LIN {X 0,Y 417.094,Z 395.374,A -85,B 0,C 180,E1 -10165.652,E2 -10165.652} C_VEL
LIN {X 0,Y 417.167,Z 397.871,A -85,B 0,C 180,E1 -10167.103,E2 -10167.103} C_VEL
LIN {X 0,Y 417.136,Z 398.972,A -85,B 0,C 180,E1 -10168.069,E2 -10168.069} C_VEL
LIN {X 0,Y 417.115,Z 399.643,A -85,B 0,C 180,E1 -10169.035,E2 -10169.035} C_VEL
LIN {X 0,Y 417.13,Z 399.91,A -85,B 0,C 180,E1 -10170,E2 -10170} C_VEL
LIN {X 0,Y 417.089,Z 399.765,A -85,B 0,C 180,E1 -10170.966,E2 -10170.966} C_VEL
LIN {X 0,Y 417.118,Z 399.169,A -85,B 0,C 180,E1 -10171.931,E2 -10171.931} C_VEL
LIN {X 0,Y 417.132,Z 398.154,A -85,B 0,C 180,E1 -10172.898,E2 -10172.898} C_VEL
LIN {X 0,Y 417.056,Z 396.723,A -85,B 0,C 180,E1 -10173.865,E2 -10173.865} C_VEL
LIN {X 0,Y 417.128,Z 393.73,A -85,B 0,C 180,E1 -10175.317,E2 -10175.317} C_VEL
LIN {X 0,Y 417.159,Z 389.667,A -85,B 0,C 180,E1 -10176.773,E2 -10176.773} C_VEL
LIN {X 0,Y 417.432,Z 383.444,A -85,B 0,C 180,E1 -10178.472,E2 -10178.472} C_VEL
LIN {X 0,Y 417.77,Z 376.616,A -85,B 0,C 180,E1 -10179.93,E2 -10179.93} C_VEL
LIN {X 0,Y 418.327,Z 368.161,A -85,B 0,C 180,E1 -10181.385,E2 -10181.385} C_VEL
LIN {X 0,Y 418.871,Z 359.55,A -85,B 0,C 180,E1 -10182.599,E2 -10182.599} C_VEL
LIN {X 0,Y 419.553,Z 349.191,A -85,B 0,C 180,E1 -10183.785,E2 -10183.785} C_VEL
LIN {X 0,Y 420.452,Z 337.073,A -85,B 0,C 180,E1 -10184.892,E2 -10184.892} C_VEL
LIN {X 0,Y 421.245,Z 325.274,A -85,B 0,C 180,E1 -10185.731,E2 -10185.731} C_VEL
LIN {X 0,Y 422,Z 311.923,A -85,B 0,C 180,E1 -10186.447,E2 -10186.447} C_VEL
LIN {X 0,Y 422.679,Z 299.417,A -85,B 0,C 180,E1 -10186.917,E2 -10186.917} C_VEL
LIN {X 0,Y 423.066,Z 283.977,A -85,B 0,C 180,E1 -10187.274,E2 -10187.274} C_VEL
LIN {X 0,Y 424.143,Z 213.784,A -85,B 0,C 180,E1 -10188.664,E2 -10188.664} C_VEL
LIN {X 0,Y 421.797,Z 196.296,A -85,B 0,C 180,E1 -10189.167,E2 -10189.167} C_VEL
LIN {X 0,Y 419.76,Z 184.639,A -85,B 0,C 180,E1 -10189.564,E2 -10189.564} C_VEL
LIN {X 0,Y 421.003,Z 163.827,A -85,B 0,C 180,E1 -10193.343,E2 -10193.343} C_VEL
LIN {X 0,Y 421.708,Z 152.632,A -85,B 0,C 180,E1 -10195.413,E2 -10195.413} C_VEL
LIN {X 0,Y 419.796,Z 142.649,A -85,B 0,C 180,E1 -10197.464,E2 -10197.464} C_VEL
LIN {X 0,Y 418.315,Z 136.387,A -85,B 0,C 180,E1 -10198.855,E2 -10198.855} C_VEL
LIN {X 0,Y 418.249,Z 136.39,A -85,B 0,C 180,E1 -10202.528,E2 -10202.528} C_VEL
LIN {X 0,Y 418.263,Z 136.385,A -85,B 0,C 180,E1 -10204.841,E2 -10204.841} C_VEL
LIN {X 0,Y 418.261,Z 136.386,A -85,B 0,C 180,E1 -10208.441,E2 -10208.441} C_VEL
LIN {X 0,Y 418.227,Z 136.388,A -85,B 0,C 180,E1 -10210.948,E2 -10210.948} C_VEL
LIN {X 0,Y 418.214,Z 136.391,A -85,B 0,C 180,E1 -10213.729,E2 -10213.729} C_VEL
LIN {X 0,Y 418.213,Z 136.388,A -85,B 0,C 180,E1 -10216.449,E2 -10216.449} C_VEL
LIN {X 0,Y 418.226,Z 136.384,A -85,B 0,C 180,E1 -10219.13,E2 -10219.13} C_VEL
LIN {X 0,Y 418.229,Z 136.385,A -85,B 0,C 180,E1 -10222.167,E2 -10222.167} C_VEL
LIN {X 0,Y 418.267,Z 136.382,A -85,B 0,C 180,E1 -10225.42,E2 -10225.42} C_VEL
LIN {X 0,Y 418.214,Z 136.384,A -85,B 0,C 180,E1 -10228.604,E2 -10228.604} C_VEL
LIN {X 0,Y 418.295,Z 136.38,A -85,B 0,C 180,E1 -10231.937,E2 -10231.937} C_VEL
LIN {X 0,Y 418.293,Z 136.38,A -85,B 0,C 180,E1 -10235.163,E2 -10235.163} C_VEL
LIN {X 0,Y 418.237,Z 136.385,A -85,B 0,C 180,E1 -10238.303,E2 -10238.303} C_VEL
LIN {X 0,Y 418.278,Z 136.38,A -85,B 0,C 180,E1 -10241.383,E2 -10241.383} C_VEL
LIN {X 0,Y 418.304,Z 136.377,A -85,B 0,C 180,E1 -10244.406,E2 -10244.406} C_VEL
LIN {X 0,Y 418.359,Z 136.373,A -85,B 0,C 180,E1 -10247.385,E2 -10247.385} C_VEL
LIN {X 0,Y 418.341,Z 136.376,A -85,B 0,C 180,E1 -10250.328,E2 -10250.328} C_VEL
LIN {X 0,Y 418.463,Z 136.363,A -85,B 0,C 180,E1 -10253.248,E2 -10253.248} C_VEL
LIN {X 0,Y 418.336,Z 136.378,A -85,B 0,C 180,E1 -10255.181,E2 -10255.181} C_VEL
LIN {X 0,Y 418.543,Z 136.354,A -85,B 0,C 180,E1 -10258.075,E2 -10258.075} C_VEL
LIN {X 0,Y 418.669,Z 136.335,A -85,B 0,C 180,E1 -10260,E2 -10260} C_VEL
LIN {X 0,Y 418.49,Z 136.36,A -85,B 0,C 180,E1 -10262.887,E2 -10262.887} C_VEL
LIN {X 0,Y 418.393,Z 136.563,A -85,B 0,C 180,E1 -10263.43,E2 -10263.43} C_VEL
LIN {X 0,Y 420.352,Z 145.319,A -85,B 0,C 180,E1 -10265.546,E2 -10265.546} C_VEL
LIN {X 0,Y 422.812,Z 152.93,A -85,B 0,C 180,E1 -10265.873,E2 -10265.873} C_VEL
LIN {X 0,Y 425.067,Z 163.368,A -85,B 0,C 180,E1 -10266.228,E2 -10266.228} C_VEL
LIN {X 0,Y 423.251,Z 252.714,A -85,B 0,C 180,E1 -10268.023,E2 -10268.023} C_VEL
LIN {X 0,Y 422.865,Z 266.764,A -85,B 0,C 180,E1 -10268.512,E2 -10268.512} C_VEL
LIN {X 0,Y 422.412,Z 278.341,A -85,B 0,C 180,E1 -10269.094,E2 -10269.094} C_VEL
LIN {X 0,Y 421.766,Z 290.403,A -85,B 0,C 180,E1 -10269.903,E2 -10269.903} C_VEL
LIN {X 0,Y 421.007,Z 302.463,A -85,B 0,C 180,E1 -10270.946,E2 -10270.946} C_VEL
LIN {X 0,Y 420.288,Z 312.69,A -85,B 0,C 180,E1 -10272.065,E2 -10272.065} C_VEL
LIN {X 0,Y 419.627,Z 321.922,A -85,B 0,C 180,E1 -10273.314,E2 -10273.314} C_VEL
LIN {X 0,Y 419.021,Z 329.545,A -85,B 0,C 180,E1 -10274.571,E2 -10274.571} C_VEL
LIN {X 0,Y 418.437,Z 336.998,A -85,B 0,C 180,E1 -10276.089,E2 -10276.089} C_VEL
LIN {X 0,Y 418.001,Z 342.862,A -85,B 0,C 180,E1 -10277.616,E2 -10277.616} C_VEL
LIN {X 0,Y 417.659,Z 347.251,A -85,B 0,C 180,E1 -10279.083,E2 -10279.083} C_VEL
LIN {X 0,Y 417.369,Z 350.82,A -85,B 0,C 180,E1 -10280.708,E2 -10280.708} C_VEL
LIN {X 0,Y 417.184,Z 352.874,A -85,B 0,C 180,E1 -10282.097,E2 -10282.097} C_VEL
LIN {X 0,Y 417.034,Z 354.234,A -85,B 0,C 180,E1 -10283.857,E2 -10283.857} C_VEL
LIN {X 0,Y 417.033,Z 354.402,A -85,B 0,C 180,E1 -10284.917,E2 -10284.917} C_VEL
LIN {X 0,Y 417.067,Z 353.497,A -85,B 0,C 180,E1 -10286.733,E2 -10286.733} C_VEL
LIN {X 0,Y 417.126,Z 351.798,A -85,B 0,C 180,E1 -10288.148,E2 -10288.148} C_VEL
LIN {X 0,Y 417.344,Z 348.667,A -85,B 0,C 180,E1 -10289.786,E2 -10289.786} C_VEL
LIN {X 0,Y 417.543,Z 344.141,A -85,B 0,C 180,E1 -10291.452,E2 -10291.452} C_VEL
LIN {X 0,Y 417.849,Z 339.491,A -85,B 0,C 180,E1 -10292.757,E2 -10292.757} C_VEL
LIN {X 0,Y 418.25,Z 332.297,A -85,B 0,C 180,E1 -10294.364,E2 -10294.364} C_VEL
LIN {X 0,Y 418.73,Z 324.93,A -85,B 0,C 180,E1 -10295.679,E2 -10295.679} C_VEL
LIN {X 0,Y 419.225,Z 316.571,A -85,B 0,C 180,E1 -10296.906,E2 -10296.906} C_VEL
LIN {X 0,Y 419.837,Z 306.507,A -85,B 0,C 180,E1 -10298.115,E2 -10298.115} C_VEL
LIN {X 0,Y 420.414,Z 296,A -85,B 0,C 180,E1 -10299.128,E2 -10299.128} C_VEL
LIN {X 0,Y 420.983,Z 284.099,A -85,B 0,C 180,E1 -10300.04,E2 -10300.04} C_VEL
LIN {X 0,Y 421.48,Z 272.646,A -85,B 0,C 180,E1 -10300.719,E2 -10300.719} C_VEL
LIN {X 0,Y 421.837,Z 259.788,A -85,B 0,C 180,E1 -10301.279,E2 -10301.279} C_VEL
LIN {X 0,Y 422.128,Z 246.612,A -85,B 0,C 180,E1 -10301.649,E2 -10301.649} C_VEL
LIN {X 0,Y 423.408,Z 161.415,A -85,B 0,C 180,E1 -10303.267,E2 -10303.267} C_VEL
LIN {X 0,Y 419.546,Z 143.216,A -85,B 0,C 180,E1 -10303.8,E2 -10303.8} C_VEL
LIN {X 0,Y 418.289,Z 136.384,A -85,B 0,C 180,E1 -10305.466,E2 -10305.466} C_VEL
LIN {X 0,Y 418.222,Z 136.387,A -85,B 0,C 180,E1 -10309.13,E2 -10309.13} C_VEL
LIN {X 0,Y 418.225,Z 136.387,A -85,B 0,C 180,E1 -10312.167,E2 -10312.167} C_VEL
LIN {X 0,Y 418.263,Z 136.386,A -85,B 0,C 180,E1 -10315.42,E2 -10315.42} C_VEL
LIN {X 0,Y 418.21,Z 136.387,A -85,B 0,C 180,E1 -10318.603,E2 -10318.603} C_VEL
LIN {X 0,Y 418.291,Z 136.379,A -85,B 0,C 180,E1 -10321.936,E2 -10321.936} C_VEL
LIN {X 0,Y 418.289,Z 136.382,A -85,B 0,C 180,E1 -10325.162,E2 -10325.162} C_VEL
LIN {X 0,Y 418.276,Z 136.378,A -85,B 0,C 180,E1 -10326.002,E2 -10326.002} C_VEL
LIN {X 0,Y 417.636,Z 136.462,A -85,B 0,C 180,E1 -10326.805,E2 -10326.805} C_VEL
LIN {X 0,Y 414.786,Z 136.814,A -85,B 0,C 180,E1 -10328.11,E2 -10328.11} C_VEL
LIN {X 0,Y 412.35,Z 137.123,A -85,B 0,C 180,E1 -10329.164,E2 -10329.164} C_VEL
LIN {X 0,Y 411.294,Z 137.249,A -85,B 0,C 180,E1 -10329.978,E2 -10329.978} C_VEL
LIN {X 0,Y 411.204,Z 137.26,A -85,B 0,C 180,E1 -10330.254,E2 -10330.254} C_VEL
LIN {X 0,Y 411.262,Z 137.259,A -85,B 0,C 180,E1 -10333.131,E2 -10333.131} C_VEL
LIN {X 0,Y 411.304,Z 137.252,A -85,B 0,C 180,E1 -10336.895,E2 -10336.895} C_VEL
LIN {X 0,Y 411.292,Z 137.249,A -85,B 0,C 180,E1 -10340.161,E2 -10340.161} C_VEL
LIN {X 0,Y 411.45,Z 137.234,A -85,B 0,C 180,E1 -10343.133,E2 -10343.133} C_VEL
LIN {X 0,Y 411.308,Z 137.252,A -85,B 0,C 180,E1 -10345.099,E2 -10345.099} C_VEL
LIN {X 0,Y 411.513,Z 137.221,A -85,B 0,C 180,E1 -10348.042,E2 -10348.042} C_VEL
LIN {X 0,Y 411.641,Z 137.205,A -85,B 0,C 180,E1 -10350,E2 -10350} C_VEL
LIN {X 0,Y 411.463,Z 137.232,A -85,B 0,C 180,E1 -10352.937,E2 -10352.937} C_VEL
LIN {X 0,Y 411.45,Z 137.234,A -85,B 0,C 180,E1 -10356.867,E2 -10356.867} C_VEL
LIN {X 0,Y 411.291,Z 137.249,A -85,B 0,C 180,E1 -10359.838,E2 -10359.838} C_VEL
LIN {X 0,Y 411.303,Z 137.249,A -85,B 0,C 180,E1 -10363.104,E2 -10363.104} C_VEL
LIN {X 0,Y 411.26,Z 137.255,A -85,B 0,C 180,E1 -10366.869,E2 -10366.869} C_VEL
LIN {X 0,Y 411.228,Z 137.259,A -85,B 0,C 180,E1 -10369.986,E2 -10369.986} C_VEL
LIN {X 0,Y 411.193,Z 137.261,A -85,B 0,C 180,E1 -10373.148,E2 -10373.148} C_VEL
LIN {X 0,Y 411.233,Z 137.262,A -85,B 0,C 180,E1 -10376.381,E2 -10376.381} C_VEL
LIN {X 0,Y 411.208,Z 137.261,A -85,B 0,C 180,E1 -10379.712,E2 -10379.712} C_VEL
LIN {X 0,Y 411.204,Z 137.26,A -85,B 0,C 180,E1 -10383.156,E2 -10383.156} C_VEL
LIN {X 0,Y 411.192,Z 137.263,A -85,B 0,C 180,E1 -10386.553,E2 -10386.553} C_VEL
LIN {X 0,Y 411.213,Z 137.263,A -85,B 0,C 180,E1 -10389.728,E2 -10389.728} C_VEL
LIN {X 0,Y 411.227,Z 137.257,A -85,B 0,C 180,E1 -10393.126,E2 -10393.126} C_VEL
LIN {X 0,Y 411.168,Z 137.271,A -85,B 0,C 180,E1 -10395.88,E2 -10395.88} C_VEL
LIN {X 0,Y 411.208,Z 137.263,A -85,B 0,C 180,E1 -10399.499,E2 -10399.499} C_VEL
LIN {X 0,Y 411.2,Z 137.263,A -85,B 0,C 180,E1 -10402.027,E2 -10402.027} C_VEL
LIN {X 0,Y 411.203,Z 137.266,A -85,B 0,C 180,E1 -10405.667,E2 -10405.667} C_VEL
LIN {X 0,Y 411.186,Z 137.265,A -85,B 0,C 180,E1 -10409.153,E2 -10409.153} C_VEL
LIN {X 0,Y 411.255,Z 137.253,A -85,B 0,C 180,E1 -10412.523,E2 -10412.523} C_VEL
LIN {X 0,Y 411.224,Z 137.26,A -85,B 0,C 180,E1 -10415.785,E2 -10415.785} C_VEL
LIN {X 0,Y 411.193,Z 137.264,A -85,B 0,C 180,E1 -10418.966,E2 -10418.966} C_VEL
LIN {X 0,Y 411.25,Z 137.254,A -85,B 0,C 180,E1 -10422.085,E2 -10422.085} C_VEL
LIN {X 0,Y 411.257,Z 137.26,A -85,B 0,C 180,E1 -10425.148,E2 -10425.148} C_VEL
LIN {X 0,Y 411.282,Z 137.25,A -85,B 0,C 180,E1 -10428.168,E2 -10428.168} C_VEL
LIN {X 0,Y 411.438,Z 137.231,A -85,B 0,C 180,E1 -10432.189,E2 -10432.189} C_VEL
LIN {X 0,Y 411.469,Z 137.227,A -85,B 0,C 180,E1 -10434.118,E2 -10434.118} C_VEL
LIN {X 0,Y 411.512,Z 137.221,A -85,B 0,C 180,E1 -10438.043,E2 -10438.043} C_VEL
LIN {X 0,Y 411.64,Z 137.205,A -85,B 0,C 180,E1 -10440,E2 -10440} C_VEL
LIN {X 0,Y 411.463,Z 137.233,A -85,B 0,C 180,E1 -10442.938,E2 -10442.938} C_VEL
LIN {X 0,Y 411.459,Z 137.233,A -85,B 0,C 180,E1 -10446.867,E2 -10446.867} C_VEL
LIN {X 0,Y 411.292,Z 137.249,A -85,B 0,C 180,E1 -10449.839,E2 -10449.839} C_VEL
LIN {X 0,Y 411.304,Z 137.249,A -85,B 0,C 180,E1 -10453.105,E2 -10453.105} C_VEL
LIN {X 0,Y 411.262,Z 137.255,A -85,B 0,C 180,E1 -10456.869,E2 -10456.869} C_VEL
LIN {X 0,Y 411.229,Z 137.259,A -85,B 0,C 180,E1 -10459.987,E2 -10459.987} C_VEL
LIN {X 0,Y 411.194,Z 137.261,A -85,B 0,C 180,E1 -10463.148,E2 -10463.148} C_VEL
LIN {X 0,Y 411.235,Z 137.262,A -85,B 0,C 180,E1 -10466.381,E2 -10466.381} C_VEL
LIN {X 0,Y 411.199,Z 137.262,A -85,B 0,C 180,E1 -10469.713,E2 -10469.713} C_VEL
LIN {X 0,Y 411.206,Z 137.259,A -85,B 0,C 180,E1 -10473.156,E2 -10473.156} C_VEL
LIN {X 0,Y 411.195,Z 137.263,A -85,B 0,C 180,E1 -10476.554,E2 -10476.554} C_VEL
LIN {X 0,Y 411.226,Z 137.261,A -85,B 0,C 180,E1 -10479.731,E2 -10479.731} C_VEL
LIN {X 0,Y 411.178,Z 137.263,A -85,B 0,C 180,E1 -10483.133,E2 -10483.133} C_VEL
LIN {X 0,Y 411.168,Z 137.271,A -85,B 0,C 180,E1 -10485.882,E2 -10485.882} C_VEL
LIN {X 0,Y 411.163,Z 137.265,A -85,B 0,C 180,E1 -10488.772,E2 -10488.772} C_VEL
LIN {X 0,Y 411.205,Z 137.266,A -85,B 0,C 180,E1 -10491.832,E2 -10491.832} C_VEL
LIN {X 0,Y 411.211,Z 137.26,A -85,B 0,C 180,E1 -10495.122,E2 -10495.122} C_VEL
LIN {X 0,Y 411.166,Z 137.269,A -85,B 0,C 180,E1 -10498.003,E2 -10498.003} C_VEL
LIN {X 0,Y 411.299,Z 137.404,A -85,B 0,C 180,E1 -10501.326,E2 -10501.326} C_VEL
LIN {X 0,Y 414.04,Z 150.868,A -85,B 0,C 180,E1 -10504.111,E2 -10504.111} C_VEL
LIN {X 0,Y 414.425,Z 154.951,A -85,B 0,C 180,E1 -10504.916,E2 -10504.916} C_VEL
LIN {X 0,Y 413.221,Z 172.954,A -85,B 0,C 180,E1 -10508.29,E2 -10508.29} C_VEL
LIN {X 0,Y 412.419,Z 187.182,A -85,B 0,C 180,E1 -10510.923,E2 -10510.923} C_VEL
LIN {X 0,Y 416.159,Z 215.844,A -85,B 0,C 180,E1 -10511.653,E2 -10511.653} C_VEL
LIN {X 0,Y 414.934,Z 296.264,A -85,B 0,C 180,E1 -10513.234,E2 -10513.234} C_VEL
LIN {X 0,Y 414.347,Z 310.436,A -85,B 0,C 180,E1 -10513.717,E2 -10513.717} C_VEL
LIN {X 0,Y 413.746,Z 323.086,A -85,B 0,C 180,E1 -10514.357,E2 -10514.357} C_VEL
LIN {X 0,Y 412.93,Z 335.573,A -85,B 0,C 180,E1 -10515.209,E2 -10515.209} C_VEL
LIN {X 0,Y 412.315,Z 346.811,A -85,B 0,C 180,E1 -10516.195,E2 -10516.195} C_VEL
LIN {X 0,Y 411.774,Z 355.924,A -85,B 0,C 180,E1 -10517.181,E2 -10517.181} C_VEL
LIN {X 0,Y 411.231,Z 365.272,A -85,B 0,C 180,E1 -10518.416,E2 -10518.416} C_VEL
LIN {X 0,Y 410.638,Z 374.356,A -85,B 0,C 180,E1 -10519.897,E2 -10519.897} C_VEL
LIN {X 0,Y 410.346,Z 381.654,A -85,B 0,C 180,E1 -10521.381,E2 -10521.381} C_VEL
LIN {X 0,Y 410.166,Z 386.569,A -85,B 0,C 180,E1 -10522.617,E2 -10522.617} C_VEL
LIN {X 0,Y 410.009,Z 391.307,A -85,B 0,C 180,E1 -10524.097,E2 -10524.097} C_VEL
LIN {X 0,Y 410.021,Z 394.891,A -85,B 0,C 180,E1 -10525.577,E2 -10525.577} C_VEL
LIN {X 0,Y 410.08,Z 397.415,A -85,B 0,C 180,E1 -10527.053,E2 -10527.053} C_VEL
LIN {X 0,Y 410.063,Z 398.546,A -85,B 0,C 180,E1 -10528.036,E2 -10528.036} C_VEL
LIN {X 0,Y 410.034,Z 399.229,A -85,B 0,C 180,E1 -10529.018,E2 -10529.018} C_VEL
LIN {X 0,Y 410.046,Z 399.509,A -85,B 0,C 180,E1 -10530,E2 -10530} C_VEL
LIN {X 0,Y 410.01,Z 399.378,A -85,B 0,C 180,E1 -10530.983,E2 -10530.983} C_VEL
LIN {X 0,Y 410.045,Z 398.803,A -85,B 0,C 180,E1 -10531.965,E2 -10531.965} C_VEL
LIN {X 0,Y 410.029,Z 397.798,A -85,B 0,C 180,E1 -10532.948,E2 -10532.948} C_VEL
LIN {X 0,Y 409.972,Z 396.378,A -85,B 0,C 180,E1 -10533.932,E2 -10533.932} C_VEL
LIN {X 0,Y 410.018,Z 393.403,A -85,B 0,C 180,E1 -10535.41,E2 -10535.41} C_VEL
LIN {X 0,Y 410.077,Z 389.358,A -85,B 0,C 180,E1 -10536.891,E2 -10536.891} C_VEL
LIN {X 0,Y 410.355,Z 383.175,A -85,B 0,C 180,E1 -10538.619,E2 -10538.619} C_VEL
LIN {X 0,Y 410.741,Z 376.38,A -85,B 0,C 180,E1 -10540.101,E2 -10540.101} C_VEL
LIN {X 0,Y 411.335,Z 367.962,A -85,B 0,C 180,E1 -10541.582,E2 -10541.582} C_VEL
LIN {X 0,Y 411.903,Z 359.384,A -85,B 0,C 180,E1 -10542.816,E2 -10542.816} C_VEL
LIN {X 0,Y 412.662,Z 348.874,A -85,B 0,C 180,E1 -10544.046,E2 -10544.046} C_VEL
LIN {X 0,Y 413.588,Z 337.088,A -85,B 0,C 180,E1 -10545.145,E2 -10545.145} C_VEL
LIN {X 0,Y 414.44,Z 325.483,A -85,B 0,C 180,E1 -10545.996,E2 -10545.996} C_VEL
LIN {X 0,Y 415.225,Z 312.334,A -85,B 0,C 180,E1 -10546.723,E2 -10546.723} C_VEL
LIN {X 0,Y 415.967,Z 299.323,A -85,B 0,C 180,E1 -10547.23,E2 -10547.23} C_VEL
LIN {X 0,Y 416.379,Z 284.262,A -85,B 0,C 180,E1 -10547.592,E2 -10547.592} C_VEL
LIN {X 0,Y 417.533,Z 214.569,A -85,B 0,C 180,E1 -10549.008,E2 -10549.008} C_VEL
LIN {X 0,Y 415.28,Z 197.666,A -85,B 0,C 180,E1 -10549.512,E2 -10549.512} C_VEL
LIN {X 0,Y 412.933,Z 184.186,A -85,B 0,C 180,E1 -10549.976,E2 -10549.976} C_VEL
LIN {X 0,Y 414.158,Z 164.617,A -85,B 0,C 180,E1 -10553.602,E2 -10553.602} C_VEL
LIN {X 0,Y 414.86,Z 154.266,A -85,B 0,C 180,E1 -10555.546,E2 -10555.546} C_VEL
LIN {X 0,Y 412.871,Z 143.922,A -85,B 0,C 180,E1 -10557.728,E2 -10557.728} C_VEL
LIN {X 0,Y 411.237,Z 137.268,A -85,B 0,C 180,E1 -10559.211,E2 -10559.211} C_VEL
LIN {X 0,Y 411.169,Z 137.273,A -85,B 0,C 180,E1 -10561.997,E2 -10561.997} C_VEL
LIN {X 0,Y 411.214,Z 137.263,A -85,B 0,C 180,E1 -10564.879,E2 -10564.879} C_VEL
LIN {X 0,Y 411.211,Z 137.265,A -85,B 0,C 180,E1 -10568.169,E2 -10568.169} C_VEL
LIN {X 0,Y 411.168,Z 137.268,A -85,B 0,C 180,E1 -10571.228,E2 -10571.228} C_VEL
LIN {X 0,Y 411.179,Z 137.266,A -85,B 0,C 180,E1 -10574.49,E2 -10574.49} C_VEL
LIN {X 0,Y 411.181,Z 137.262,A -85,B 0,C 180,E1 -10578.195,E2 -10578.195} C_VEL
LIN {X 0,Y 411.214,Z 137.256,A -85,B 0,C 180,E1 -10580.775,E2 -10580.775} C_VEL
LIN {X 0,Y 411.2,Z 137.26,A -85,B 0,C 180,E1 -10584.471,E2 -10584.471} C_VEL
LIN {X 0,Y 411.21,Z 137.258,A -85,B 0,C 180,E1 -10586.873,E2 -10586.873} C_VEL
LIN {X 0,Y 411.236,Z 137.258,A -85,B 0,C 180,E1 -10590.644,E2 -10590.644} C_VEL
LIN {X 0,Y 411.241,Z 137.256,A -85,B 0,C 180,E1 -10593.619,E2 -10593.619} C_VEL
LIN {X 0,Y 411.206,Z 137.261,A -85,B 0,C 180,E1 -10596.852,E2 -10596.852} C_VEL
LIN {X 0,Y 411.218,Z 137.258,A -85,B 0,C 180,E1 -10600.05,E2 -10600.05} C_VEL
LIN {X 0,Y 411.266,Z 137.258,A -85,B 0,C 180,E1 -10603.131,E2 -10603.131} C_VEL
LIN {X 0,Y 411.309,Z 137.25,A -85,B 0,C 180,E1 -10606.896,E2 -10606.896} C_VEL
LIN {X 0,Y 411.294,Z 137.253,A -85,B 0,C 180,E1 -10610.161,E2 -10610.161} C_VEL
LIN {X 0,Y 411.427,Z 137.24,A -85,B 0,C 180,E1 -10613.132,E2 -10613.132} C_VEL
LIN {X 0,Y 411.307,Z 137.254,A -85,B 0,C 180,E1 -10615.099,E2 -10615.099} C_VEL
LIN {X 0,Y 411.512,Z 137.229,A -85,B 0,C 180,E1 -10618.042,E2 -10618.042} C_VEL
LIN {X 0,Y 411.638,Z 137.211,A -85,B 0,C 180,E1 -10620,E2 -10620} C_VEL
LIN {X 0,Y 411.436,Z 137.333,A -85,B 0,C 180,E1 -10623.029,E2 -10623.029} C_VEL
LIN {X 0,Y 413.317,Z 146.112,A -85,B 0,C 180,E1 -10625.136,E2 -10625.136} C_VEL
LIN {X 0,Y 416.269,Z 154.049,A -85,B 0,C 180,E1 -10625.504,E2 -10625.504} C_VEL
LIN {X 0,Y 418.496,Z 164.589,A -85,B 0,C 180,E1 -10625.873,E2 -10625.873} C_VEL
LIN {X 0,Y 416.604,Z 253.162,A -85,B 0,C 180,E1 -10627.695,E2 -10627.695} C_VEL
LIN {X 0,Y 416.181,Z 267.162,A -85,B 0,C 180,E1 -10628.191,E2 -10628.191} C_VEL
LIN {X 0,Y 415.672,Z 279.237,A -85,B 0,C 180,E1 -10628.813,E2 -10628.813} C_VEL
LIN {X 0,Y 415.007,Z 291.038,A -85,B 0,C 180,E1 -10629.626,E2 -10629.626} C_VEL
LIN {X 0,Y 414.301,Z 301.835,A -85,B 0,C 180,E1 -10630.569,E2 -10630.569} C_VEL
LIN {X 0,Y 413.533,Z 311.8,A -85,B 0,C 180,E1 -10631.643,E2 -10631.643} C_VEL
LIN {X 0,Y 412.855,Z 320.438,A -85,B 0,C 180,E1 -10632.785,E2 -10632.785} C_VEL
LIN {X 0,Y 412.205,Z 328.363,A -85,B 0,C 180,E1 -10634.061,E2 -10634.061} C_VEL
LIN {X 0,Y 411.529,Z 336.111,A -85,B 0,C 180,E1 -10635.603,E2 -10635.603} C_VEL
LIN {X 0,Y 411.114,Z 341.34,A -85,B 0,C 180,E1 -10636.894,E2 -10636.894} C_VEL
LIN {X 0,Y 410.726,Z 346.366,A -85,B 0,C 180,E1 -10638.454,E2 -10638.454} C_VEL
LIN {X 0,Y 410.413,Z 350.167,A -85,B 0,C 180,E1 -10640.028,E2 -10640.028} C_VEL
LIN {X 0,Y 410.224,Z 352.057,A -85,B 0,C 180,E1 -10641.086,E2 -10641.086} C_VEL
LIN {X 0,Y 410.107,Z 353.572,A -85,B 0,C 180,E1 -10642.271,E2 -10642.271} C_VEL
LIN {X 0,Y 410.009,Z 354.368,A -85,B 0,C 180,E1 -10643.218,E2 -10643.218} C_VEL
LIN {X 0,Y 409.956,Z 354.806,A -85,B 0,C 180,E1 -10644.687,E2 -10644.687} C_VEL
LIN {X 0,Y 409.977,Z 354.111,A -85,B 0,C 180,E1 -10646.468,E2 -10646.468} C_VEL
LIN {X 0,Y 410.004,Z 352.991,A -85,B 0,C 180,E1 -10647.568,E2 -10647.568} C_VEL
LIN {X 0,Y 410.18,Z 350.577,A -85,B 0,C 180,E1 -10649.093,E2 -10649.093} C_VEL
LIN {X 0,Y 410.412,Z 346.305,A -85,B 0,C 180,E1 -10650.912,E2 -10650.912} C_VEL
LIN {X 0,Y 410.703,Z 340.963,A -85,B 0,C 180,E1 -10652.548,E2 -10652.548} C_VEL
LIN {X 0,Y 411.088,Z 334.692,A -85,B 0,C 180,E1 -10654.048,E2 -10654.048} C_VEL
LIN {X 0,Y 411.592,Z 327.195,A -85,B 0,C 180,E1 -10655.489,E2 -10655.489} C_VEL
LIN {X 0,Y 412.144,Z 317.944,A -85,B 0,C 180,E1 -10656.917,E2 -10656.917} C_VEL
LIN {X 0,Y 412.8,Z 307.838,A -85,B 0,C 180,E1 -10658.171,E2 -10658.171} C_VEL
LIN {X 0,Y 413.444,Z 296.645,A -85,B 0,C 180,E1 -10659.286,E2 -10659.286} C_VEL
LIN {X 0,Y 414.011,Z 285.124,A -85,B 0,C 180,E1 -10660.191,E2 -10660.191} C_VEL
LIN {X 0,Y 414.577,Z 272.727,A -85,B 0,C 180,E1 -10660.943,E2 -10660.943} C_VEL
LIN {X 0,Y 414.931,Z 259.918,A -85,B 0,C 180,E1 -10661.505,E2 -10661.505} C_VEL
LIN {X 0,Y 415.256,Z 246.295,A -85,B 0,C 180,E1 -10661.888,E2 -10661.888} C_VEL
LIN {X 0,Y 416.505,Z 161.872,A -85,B 0,C 180,E1 -10663.527,E2 -10663.527} C_VEL
LIN {X 0,Y 412.883,Z 145.219,A -85,B 0,C 180,E1 -10664.014,E2 -10664.014} C_VEL
LIN {X 0,Y 412.442,Z 143.564,A -85,B 0,C 180,E1 -10664.082,E2 -10664.082} C_VEL
LIN {X 0,Y 411.254,Z 137.26,A -85,B 0,C 180,E1 -10665.629,E2 -10665.629} C_VEL
LIN {X 0,Y 411.179,Z 137.268,A -85,B 0,C 180,E1 -10669.495,E2 -10669.495} C_VEL
LIN {X 0,Y 411.191,Z 137.264,A -85,B 0,C 180,E1 -10672.026,E2 -10672.026} C_VEL
LIN {X 0,Y 411.204,Z 137.265,A -85,B 0,C 180,E1 -10675.666,E2 -10675.666} C_VEL
LIN {X 0,Y 411.189,Z 137.265,A -85,B 0,C 180,E1 -10679.152,E2 -10679.152} C_VEL
LIN {X 0,Y 411.258,Z 137.253,A -85,B 0,C 180,E1 -10682.522,E2 -10682.522} C_VEL
LIN {X 0,Y 411.21,Z 137.26,A -85,B 0,C 180,E1 -10685.993,E2 -10685.993} C_VEL
LIN {X 0,Y 411.195,Z 137.264,A -85,B 0,C 180,E1 -10688.966,E2 -10688.966} C_VEL
LIN {X 0,Y 411.204,Z 137.26,A -85,B 0,C 180,E1 -10690.254,E2 -10690.254} C_VEL
LIN {X 0,Y 410.528,Z 137.349,A -85,B 0,C 180,E1 -10691.073,E2 -10691.073} C_VEL
LIN {X 0,Y 407.683,Z 137.699,A -85,B 0,C 180,E1 -10692.403,E2 -10692.403} C_VEL
LIN {X 0,Y 405.289,Z 138,A -85,B 0,C 180,E1 -10693.477,E2 -10693.477} C_VEL
LIN {X 0,Y 404.273,Z 138.124,A -85,B 0,C 180,E1 -10694.307,E2 -10694.307} C_VEL
LIN {X 0,Y 404.196,Z 138.134,A -85,B 0,C 180,E1 -10694.588,E2 -10694.588} C_VEL
LIN {X 0,Y 404.256,Z 138.125,A -85,B 0,C 180,E1 -10697.958,E2 -10697.958} C_VEL
LIN {X 0,Y 404.403,Z 138.107,A -85,B 0,C 180,E1 -10702.129,E2 -10702.129} C_VEL
LIN {X 0,Y 404.418,Z 138.105,A -85,B 0,C 180,E1 -10704.015,E2 -10704.015} C_VEL
LIN {X 0,Y 404.482,Z 138.097,A -85,B 0,C 180,E1 -10708.008,E2 -10708.008} C_VEL
LIN {X 0,Y 404.61,Z 138.081,A -85,B 0,C 180,E1 -10710,E2 -10710} C_VEL
LIN {X 0,Y 404.42,Z 138.109,A -85,B 0,C 180,E1 -10712.988,E2 -10712.988} C_VEL
LIN {X 0,Y 404.397,Z 138.111,A -85,B 0,C 180,E1 -10716.987,E2 -10716.987} C_VEL
LIN {X 0,Y 404.257,Z 138.126,A -85,B 0,C 180,E1 -10720.011,E2 -10720.011} C_VEL
LIN {X 0,Y 404.264,Z 138.125,A -85,B 0,C 180,E1 -10723.211,E2 -10723.211} C_VEL
LIN {X 0,Y 404.213,Z 138.132,A -85,B 0,C 180,E1 -10727.007,E2 -10727.007} C_VEL
LIN {X 0,Y 404.184,Z 138.141,A -85,B 0,C 180,E1 -10730.35,E2 -10730.35} C_VEL
LIN {X 0,Y 404.16,Z 138.138,A -85,B 0,C 180,E1 -10733.575,E2 -10733.575} C_VEL
LIN {X 0,Y 404.18,Z 138.137,A -85,B 0,C 180,E1 -10735.766,E2 -10735.766} C_VEL
LIN {X 0,Y 404.195,Z 138.137,A -85,B 0,C 180,E1 -10737.999,E2 -10737.999} C_VEL
LIN {X 0,Y 404.143,Z 138.141,A -85,B 0,C 180,E1 -10741.559,E2 -10741.559} C_VEL
LIN {X 0,Y 404.182,Z 138.134,A -85,B 0,C 180,E1 -10745.016,E2 -10745.016} C_VEL
LIN {X 0,Y 404.155,Z 138.138,A -85,B 0,C 180,E1 -10748.756,E2 -10748.756} C_VEL
LIN {X 0,Y 404.185,Z 138.138,A -85,B 0,C 180,E1 -10751.61,E2 -10751.61} C_VEL
LIN {X 0,Y 404.189,Z 138.134,A -85,B 0,C 180,E1 -10754.529,E2 -10754.529} C_VEL
LIN {X 0,Y 404.167,Z 138.138,A -85,B 0,C 180,E1 -10757.3,E2 -10757.3} C_VEL
LIN {X 0,Y 404.165,Z 138.141,A -85,B 0,C 180,E1 -10759.955,E2 -10759.955} C_VEL
LIN {X 0,Y 404.136,Z 138.142,A -85,B 0,C 180,E1 -10763.124,E2 -10763.124} C_VEL
LIN {X 0,Y 404.141,Z 138.141,A -85,B 0,C 180,E1 -10766.188,E2 -10766.188} C_VEL
LIN {X 0,Y 404.142,Z 138.144,A -85,B 0,C 180,E1 -10769.715,E2 -10769.715} C_VEL
LIN {X 0,Y 404.192,Z 138.136,A -85,B 0,C 180,E1 -10773.123,E2 -10773.123} C_VEL
LIN {X 0,Y 404.175,Z 138.142,A -85,B 0,C 180,E1 -10775.335,E2 -10775.335} C_VEL
LIN {X 0,Y 404.136,Z 138.141,A -85,B 0,C 180,E1 -10778.581,E2 -10778.581} C_VEL
LIN {X 0,Y 404.208,Z 138.133,A -85,B 0,C 180,E1 -10781.762,E2 -10781.762} C_VEL
LIN {X 0,Y 404.203,Z 138.135,A -85,B 0,C 180,E1 -10784.882,E2 -10784.882} C_VEL
LIN {X 0,Y 404.254,Z 138.126,A -85,B 0,C 180,E1 -10787.959,E2 -10787.959} C_VEL
LIN {X 0,Y 404.402,Z 138.107,A -85,B 0,C 180,E1 -10792.129,E2 -10792.129} C_VEL
LIN {X 0,Y 404.417,Z 138.105,A -85,B 0,C 180,E1 -10794.015,E2 -10794.015} C_VEL
LIN {X 0,Y 404.481,Z 138.097,A -85,B 0,C 180,E1 -10798.009,E2 -10798.009} C_VEL
LIN {X 0,Y 404.61,Z 138.081,A -85,B 0,C 180,E1 -10800,E2 -10800} C_VEL
LIN {X 0,Y 404.42,Z 138.11,A -85,B 0,C 180,E1 -10802.989,E2 -10802.989} C_VEL
LIN {X 0,Y 404.41,Z 138.11,A -85,B 0,C 180,E1 -10806.988,E2 -10806.988} C_VEL
LIN {X 0,Y 404.257,Z 138.126,A -85,B 0,C 180,E1 -10810.012,E2 -10810.012} C_VEL
LIN {X 0,Y 404.265,Z 138.125,A -85,B 0,C 180,E1 -10813.212,E2 -10813.212} C_VEL
LIN {X 0,Y 404.214,Z 138.132,A -85,B 0,C 180,E1 -10817.007,E2 -10817.007} C_VEL
LIN {X 0,Y 404.186,Z 138.14,A -85,B 0,C 180,E1 -10820.351,E2 -10820.351} C_VEL
LIN {X 0,Y 404.162,Z 138.137,A -85,B 0,C 180,E1 -10823.575,E2 -10823.575} C_VEL
LIN {X 0,Y 404.182,Z 138.136,A -85,B 0,C 180,E1 -10825.767,E2 -10825.767} C_VEL
LIN {X 0,Y 404.194,Z 138.137,A -85,B 0,C 180,E1 -10828,E2 -10828} C_VEL
LIN {X 0,Y 404.138,Z 138.141,A -85,B 0,C 180,E1 -10831.559,E2 -10831.559} C_VEL
LIN {X 0,Y 404.184,Z 138.134,A -85,B 0,C 180,E1 -10835.017,E2 -10835.017} C_VEL
LIN {X 0,Y 404.162,Z 138.137,A -85,B 0,C 180,E1 -10838.757,E2 -10838.757} C_VEL
LIN {X 0,Y 404.15,Z 138.141,A -85,B 0,C 180,E1 -10841.605,E2 -10841.605} C_VEL
LIN {X 0,Y 404.147,Z 138.14,A -85,B 0,C 180,E1 -10844.523,E2 -10844.523} C_VEL
LIN {X 0,Y 404.137,Z 138.141,A -85,B 0,C 180,E1 -10847.296,E2 -10847.296} C_VEL
LIN {X 0,Y 404.169,Z 138.141,A -85,B 0,C 180,E1 -10849.956,E2 -10849.956} C_VEL
LIN {X 0,Y 404.137,Z 138.141,A -85,B 0,C 180,E1 -10853.126,E2 -10853.126} C_VEL
LIN {X 0,Y 404.146,Z 138.141,A -85,B 0,C 180,E1 -10856.188,E2 -10856.188} C_VEL
LIN {X 0,Y 404.147,Z 138.144,A -85,B 0,C 180,E1 -10859.715,E2 -10859.715} C_VEL
LIN {X 0,Y 404.227,Z 138.213,A -85,B 0,C 180,E1 -10861.083,E2 -10861.083} C_VEL
LIN {X 0,Y 407.119,Z 152.373,A -85,B 0,C 180,E1 -10864.057,E2 -10864.057} C_VEL
LIN {X 0,Y 407.411,Z 157.112,A -85,B 0,C 180,E1 -10864.999,E2 -10864.999} C_VEL
LIN {X 0,Y 406.15,Z 175.09,A -85,B 0,C 180,E1 -10868.426,E2 -10868.426} C_VEL
LIN {X 0,Y 405.477,Z 186.936,A -85,B 0,C 180,E1 -10870.641,E2 -10870.641} C_VEL
LIN {X 0,Y 409.308,Z 216.301,A -85,B 0,C 180,E1 -10871.406,E2 -10871.406} C_VEL
LIN {X 0,Y 408.038,Z 295.995,A -85,B 0,C 180,E1 -10873.007,E2 -10873.007} C_VEL
LIN {X 0,Y 407.422,Z 310.107,A -85,B 0,C 180,E1 -10873.496,E2 -10873.496} C_VEL
LIN {X 0,Y 406.81,Z 322.738,A -85,B 0,C 180,E1 -10874.147,E2 -10874.147} C_VEL
LIN {X 0,Y 406.031,Z 334.426,A -85,B 0,C 180,E1 -10874.952,E2 -10874.952} C_VEL
LIN {X 0,Y 405.364,Z 345.803,A -85,B 0,C 180,E1 -10875.953,E2 -10875.953} C_VEL
LIN {X 0,Y 404.739,Z 356.071,A -85,B 0,C 180,E1 -10877.082,E2 -10877.082} C_VEL
LIN {X 0,Y 404.097,Z 366.156,A -85,B 0,C 180,E1 -10878.463,E2 -10878.463} C_VEL
LIN {X 0,Y 403.516,Z 375.016,A -85,B 0,C 180,E1 -10879.97,E2 -10879.97} C_VEL
LIN {X 0,Y 403.261,Z 382.073,A -85,B 0,C 180,E1 -10881.481,E2 -10881.481} C_VEL
LIN {X 0,Y 403.033,Z 387.697,A -85,B 0,C 180,E1 -10882.989,E2 -10882.989} C_VEL
LIN {X 0,Y 402.94,Z 392.08,A -85,B 0,C 180,E1 -10884.496,E2 -10884.496} C_VEL
LIN {X 0,Y 402.905,Z 395.339,A -85,B 0,C 180,E1 -10885.999,E2 -10885.999} C_VEL
LIN {X 0,Y 402.98,Z 396.949,A -85,B 0,C 180,E1 -10887.001,E2 -10887.001} C_VEL
LIN {X 0,Y 402.991,Z 398.114,A -85,B 0,C 180,E1 -10888.002,E2 -10888.002} C_VEL
LIN {X 0,Y 402.957,Z 398.813,A -85,B 0,C 180,E1 -10889.001,E2 -10889.001} C_VEL
LIN {X 0,Y 402.964,Z 399.106,A -85,B 0,C 180,E1 -10890,E2 -10890} C_VEL
LIN {X 0,Y 402.934,Z 398.989,A -85,B 0,C 180,E1 -10891,E2 -10891} C_VEL
LIN {X 0,Y 402.973,Z 398.44,A -85,B 0,C 180,E1 -10891.999,E2 -10891.999} C_VEL
LIN {X 0,Y 402.927,Z 397.443,A -85,B 0,C 180,E1 -10893,E2 -10893} C_VEL
LIN {X 0,Y 402.89,Z 396.037,A -85,B 0,C 180,E1 -10894.001,E2 -10894.001} C_VEL
LIN {X 0,Y 402.908,Z 393.086,A -85,B 0,C 180,E1 -10895.506,E2 -10895.506} C_VEL
LIN {X 0,Y 403.003,Z 389.07,A -85,B 0,C 180,E1 -10897.012,E2 -10897.012} C_VEL
LIN {X 0,Y 403.304,Z 382.925,A -85,B 0,C 180,E1 -10898.771,E2 -10898.771} C_VEL
LIN {X 0,Y 403.689,Z 376.163,A -85,B 0,C 180,E1 -10900.28,E2 -10900.28} C_VEL
LIN {X 0,Y 404.349,Z 367.791,A -85,B 0,C 180,E1 -10901.785,E2 -10901.785} C_VEL
LIN {X 0,Y 404.928,Z 359.267,A -85,B 0,C 180,E1 -10903.04,E2 -10903.04} C_VEL
LIN {X 0,Y 405.777,Z 348.844,A -85,B 0,C 180,E1 -10904.289,E2 -10904.289} C_VEL
LIN {X 0,Y 406.727,Z 337.154,A -85,B 0,C 180,E1 -10905.407,E2 -10905.407} C_VEL
LIN {X 0,Y 407.647,Z 325.73,A -85,B 0,C 180,E1 -10906.27,E2 -10906.27} C_VEL
LIN {X 0,Y 408.474,Z 312.861,A -85,B 0,C 180,E1 -10907.008,E2 -10907.008} C_VEL
LIN {X 0,Y 409.27,Z 299.414,A -85,B 0,C 180,E1 -10907.553,E2 -10907.553} C_VEL
LIN {X 0,Y 409.701,Z 284.807,A -85,B 0,C 180,E1 -10907.921,E2 -10907.921} C_VEL
LIN {X 0,Y 411.046,Z 216.068,A -85,B 0,C 180,E1 -10909.347,E2 -10909.347} C_VEL
LIN {X 0,Y 408.812,Z 199.115,A -85,B 0,C 180,E1 -10909.864,E2 -10909.864} C_VEL
LIN {X 0,Y 406.121,Z 183.741,A -85,B 0,C 180,E1 -10910.408,E2 -10910.408} C_VEL
LIN {X 0,Y 407.398,Z 164.343,A -85,B 0,C 180,E1 -10914.071,E2 -10914.071} C_VEL
LIN {X 0,Y 407.998,Z 155.476,A -85,B 0,C 180,E1 -10915.783,E2 -10915.783} C_VEL
LIN {X 0,Y 405.935,Z 145.249,A -85,B 0,C 180,E1 -10917.997,E2 -10917.997} C_VEL
LIN {X 0,Y 404.165,Z 138.149,A -85,B 0,C 180,E1 -10919.661,E2 -10919.661} C_VEL
LIN {X 0,Y 404.174,Z 138.14,A -85,B 0,C 180,E1 -10923.42,E2 -10923.42} C_VEL
LIN {X 0,Y 404.145,Z 138.147,A -85,B 0,C 180,E1 -10926.246,E2 -10926.246} C_VEL
LIN {X 0,Y 404.161,Z 138.142,A -85,B 0,C 180,E1 -10928.757,E2 -10928.757} C_VEL
LIN {X 0,Y 404.127,Z 138.147,A -85,B 0,C 180,E1 -10931.6,E2 -10931.6} C_VEL
LIN {X 0,Y 404.149,Z 138.142,A -85,B 0,C 180,E1 -10934.522,E2 -10934.522} C_VEL
LIN {X 0,Y 404.14,Z 138.142,A -85,B 0,C 180,E1 -10937.296,E2 -10937.296} C_VEL
LIN {X 0,Y 404.172,Z 138.137,A -85,B 0,C 180,E1 -10939.955,E2 -10939.955} C_VEL
LIN {X 0,Y 404.139,Z 138.139,A -85,B 0,C 180,E1 -10943.125,E2 -10943.125} C_VEL
LIN {X 0,Y 404.147,Z 138.137,A -85,B 0,C 180,E1 -10946.188,E2 -10946.188} C_VEL
LIN {X 0,Y 404.149,Z 138.144,A -85,B 0,C 180,E1 -10949.715,E2 -10949.715} C_VEL
LIN {X 0,Y 404.199,Z 138.139,A -85,B 0,C 180,E1 -10953.123,E2 -10953.123} C_VEL
LIN {X 0,Y 404.181,Z 138.14,A -85,B 0,C 180,E1 -10955.334,E2 -10955.334} C_VEL
LIN {X 0,Y 404.142,Z 138.143,A -85,B 0,C 180,E1 -10958.58,E2 -10958.58} C_VEL
LIN {X 0,Y 404.207,Z 138.129,A -85,B 0,C 180,E1 -10961.761,E2 -10961.761} C_VEL
LIN {X 0,Y 404.208,Z 138.134,A -85,B 0,C 180,E1 -10964.882,E2 -10964.882} C_VEL
LIN {X 0,Y 404.259,Z 138.128,A -85,B 0,C 180,E1 -10967.958,E2 -10967.958} C_VEL
LIN {X 0,Y 404.269,Z 138.129,A -85,B 0,C 180,E1 -10970.998,E2 -10970.998} C_VEL
LIN {X 0,Y 404.396,Z 138.115,A -85,B 0,C 180,E1 -10974.014,E2 -10974.014} C_VEL
LIN {X 0,Y 404.481,Z 138.105,A -85,B 0,C 180,E1 -10978.008,E2 -10978.008} C_VEL
LIN {X 0,Y 404.608,Z 138.087,A -85,B 0,C 180,E1 -10980,E2 -10980} C_VEL
LIN {X 0,Y 404.428,Z 138.218,A -85,B 0,C 180,E1 -10982.614,E2 -10982.614} C_VEL
LIN {X 0,Y 406.153,Z 146.451,A -85,B 0,C 180,E1 -10984.668,E2 -10984.668} C_VEL
LIN {X 0,Y 409.972,Z 156.057,A -85,B 0,C 180,E1 -10985.147,E2 -10985.147} C_VEL
LIN {X 0,Y 411.93,Z 164.739,A -85,B 0,C 180,E1 -10985.476,E2 -10985.476} C_VEL
LIN {X 0,Y 409.988,Z 253.688,A -85,B 0,C 180,E1 -10987.355,E2 -10987.355} C_VEL
LIN {X 0,Y 409.524,Z 267.666,A -85,B 0,C 180,E1 -10987.86,E2 -10987.86} C_VEL
LIN {X 0,Y 408.964,Z 280.213,A -85,B 0,C 180,E1 -10988.523,E2 -10988.523} C_VEL
LIN {X 0,Y 408.179,Z 292.73,A -85,B 0,C 180,E1 -10989.414,E2 -10989.414} C_VEL
LIN {X 0,Y 407.377,Z 304.22,A -85,B 0,C 180,E1 -10990.467,E2 -10990.467} C_VEL
LIN {X 0,Y 406.481,Z 315.01,A -85,B 0,C 180,E1 -10991.721,E2 -10991.721} C_VEL
LIN {X 0,Y 405.74,Z 323.984,A -85,B 0,C 180,E1 -10993.013,E2 -10993.013} C_VEL
LIN {X 0,Y 405.099,Z 331.394,A -85,B 0,C 180,E1 -10994.313,E2 -10994.313} C_VEL
LIN {X 0,Y 404.408,Z 338.611,A -85,B 0,C 180,E1 -10995.885,E2 -10995.885} C_VEL
LIN {X 0,Y 404.018,Z 343.469,A -85,B 0,C 180,E1 -10997.2,E2 -10997.2} C_VEL
LIN {X 0,Y 403.595,Z 348.088,A -85,B 0,C 180,E1 -10998.793,E2 -10998.793} C_VEL
LIN {X 0,Y 403.261,Z 351.514,A -85,B 0,C 180,E1 -11000.399,E2 -11000.399} C_VEL
LIN {X 0,Y 403.091,Z 353.186,A -85,B 0,C 180,E1 -11001.477,E2 -11001.477} C_VEL
LIN {X 0,Y 402.986,Z 354.337,A -85,B 0,C 180,E1 -11002.561,E2 -11002.561} C_VEL
LIN {X 0,Y 402.898,Z 355.006,A -85,B 0,C 180,E1 -11003.653,E2 -11003.653} C_VEL
LIN {X 0,Y 402.854,Z 355.188,A -85,B 0,C 180,E1 -11004.883,E2 -11004.883} C_VEL
LIN {X 0,Y 402.845,Z 354.867,A -85,B 0,C 180,E1 -11005.858,E2 -11005.858} C_VEL
LIN {X 0,Y 402.892,Z 353.851,A -85,B 0,C 180,E1 -11007.172,E2 -11007.172} C_VEL
LIN {X 0,Y 402.951,Z 352.678,A -85,B 0,C 180,E1 -11008.093,E2 -11008.093} C_VEL
LIN {X 0,Y 403.194,Z 349.533,A -85,B 0,C 180,E1 -11009.807,E2 -11009.807} C_VEL
LIN {X 0,Y 403.388,Z 345.076,A -85,B 0,C 180,E1 -11011.511,E2 -11011.511} C_VEL
LIN {X 0,Y 403.753,Z 339.909,A -85,B 0,C 180,E1 -11013.008,E2 -11013.008} C_VEL
LIN {X 0,Y 404.096,Z 333.835,A -85,B 0,C 180,E1 -11014.418,E2 -11014.418} C_VEL
LIN {X 0,Y 404.679,Z 325.902,A -85,B 0,C 180,E1 -11015.897,E2 -11015.897} C_VEL
LIN {X 0,Y 405.291,Z 316.119,A -85,B 0,C 180,E1 -11017.367,E2 -11017.367} C_VEL
LIN {X 0,Y 405.939,Z 306.278,A -85,B 0,C 180,E1 -11018.555,E2 -11018.555} C_VEL
LIN {X 0,Y 406.608,Z 295.409,A -85,B 0,C 180,E1 -11019.61,E2 -11019.61} C_VEL
LIN {X 0,Y 407.177,Z 283.8,A -85,B 0,C 180,E1 -11020.51,E2 -11020.51} C_VEL
LIN {X 0,Y 407.743,Z 271.326,A -85,B 0,C 180,E1 -11021.245,E2 -11021.245} C_VEL
LIN {X 0,Y 408.074,Z 258.213,A -85,B 0,C 180,E1 -11021.802,E2 -11021.802} C_VEL
LIN {X 0,Y 408.421,Z 245.141,A -85,B 0,C 180,E1 -11022.152,E2 -11022.152} C_VEL
LIN {X 0,Y 409.775,Z 163.207,A -85,B 0,C 180,E1 -11023.771,E2 -11023.771} C_VEL
LIN {X 0,Y 406.371,Z 147.476,A -85,B 0,C 180,E1 -11024.241,E2 -11024.241} C_VEL
LIN {X 0,Y 405.32,Z 143.945,A -85,B 0,C 180,E1 -11024.367,E2 -11024.367} C_VEL
LIN {X 0,Y 404.197,Z 138.139,A -85,B 0,C 180,E1 -11025.834,E2 -11025.834} C_VEL
LIN {X 0,Y 404.168,Z 138.14,A -85,B 0,C 180,E1 -11029.955,E2 -11029.955} C_VEL
LIN {X 0,Y 404.135,Z 138.142,A -85,B 0,C 180,E1 -11033.125,E2 -11033.125} C_VEL
LIN {X 0,Y 404.144,Z 138.14,A -85,B 0,C 180,E1 -11036.187,E2 -11036.187} C_VEL
LIN {X 0,Y 404.145,Z 138.143,A -85,B 0,C 180,E1 -11039.714,E2 -11039.714} C_VEL
LIN {X 0,Y 404.195,Z 138.137,A -85,B 0,C 180,E1 -11043.122,E2 -11043.122} C_VEL
LIN {X 0,Y 404.177,Z 138.142,A -85,B 0,C 180,E1 -11045.334,E2 -11045.334} C_VEL
LIN {X 0,Y 404.138,Z 138.141,A -85,B 0,C 180,E1 -11048.58,E2 -11048.58} C_VEL
LIN {X 0,Y 404.204,Z 138.133,A -85,B 0,C 180,E1 -11051.761,E2 -11051.761} C_VEL
LIN {X 0,Y 404.196,Z 138.134,A -85,B 0,C 180,E1 -11054.588,E2 -11054.588} C_VEL
LIN {X 0,Y 403.548,Z 138.221,A -85,B 0,C 180,E1 -11055.42,E2 -11055.42} C_VEL
LIN {X 0,Y 400.718,Z 138.577,A -85,B 0,C 180,E1 -11056.772,E2 -11056.772} C_VEL
LIN {X 0,Y 398.313,Z 138.874,A -85,B 0,C 180,E1 -11057.865,E2 -11057.865} C_VEL
LIN {X 0,Y 397.277,Z 138.998,A -85,B 0,C 180,E1 -11058.709,E2 -11058.709} C_VEL
LIN {X 0,Y 397.191,Z 139.007,A -85,B 0,C 180,E1 -11058.995,E2 -11058.995} C_VEL
LIN {X 0,Y 397.36,Z 138.984,A -85,B 0,C 180,E1 -11062.075,E2 -11062.075} C_VEL
LIN {X 0,Y 397.252,Z 139.005,A -85,B 0,C 180,E1 -11064.925,E2 -11064.925} C_VEL
LIN {X 0,Y 397.451,Z 138.973,A -85,B 0,C 180,E1 -11067.973,E2 -11067.973} C_VEL
LIN {X 0,Y 397.579,Z 138.957,A -85,B 0,C 180,E1 -11070,E2 -11070} C_VEL
LIN {X 0,Y 397.379,Z 138.986,A -85,B 0,C 180,E1 -11073.041,E2 -11073.041} C_VEL
LIN {X 0,Y 397.369,Z 138.984,A -85,B 0,C 180,E1 -11076.091,E2 -11076.091} C_VEL
LIN {X 0,Y 397.251,Z 138.999,A -85,B 0,C 180,E1 -11079.161,E2 -11079.161} C_VEL
LIN {X 0,Y 397.217,Z 139.006,A -85,B 0,C 180,E1 -11082.258,E2 -11082.258} C_VEL
LIN {X 0,Y 397.177,Z 139.007,A -85,B 0,C 180,E1 -11085.392,E2 -11085.392} C_VEL
LIN {X 0,Y 397.16,Z 139.014,A -85,B 0,C 180,E1 -11088.573,E2 -11088.573} C_VEL
LIN {X 0,Y 397.093,Z 139.019,A -85,B 0,C 180,E1 -11091.818,E2 -11091.818} C_VEL
LIN {X 0,Y 397.149,Z 139.011,A -85,B 0,C 180,E1 -11095.512,E2 -11095.512} C_VEL
LIN {X 0,Y 397.124,Z 139.017,A -85,B 0,C 180,E1 -11098.543,E2 -11098.543} C_VEL
LIN {X 0,Y 397.108,Z 139.022,A -85,B 0,C 180,E1 -11102.068,E2 -11102.068} C_VEL
LIN {X 0,Y 397.117,Z 139.016,A -85,B 0,C 180,E1 -11105.503,E2 -11105.503} C_VEL
LIN {X 0,Y 397.129,Z 139.013,A -85,B 0,C 180,E1 -11108.862,E2 -11108.862} C_VEL
LIN {X 0,Y 397.155,Z 139.013,A -85,B 0,C 180,E1 -11112.255,E2 -11112.255} C_VEL
LIN {X 0,Y 397.108,Z 139.016,A -85,B 0,C 180,E1 -11115.065,E2 -11115.065} C_VEL
LIN {X 0,Y 397.106,Z 139.02,A -85,B 0,C 180,E1 -11118.014,E2 -11118.014} C_VEL
LIN {X 0,Y 397.133,Z 139.014,A -85,B 0,C 180,E1 -11121.137,E2 -11121.137} C_VEL
LIN {X 0,Y 397.116,Z 139.015,A -85,B 0,C 180,E1 -11124.497,E2 -11124.497} C_VEL
LIN {X 0,Y 397.075,Z 139.023,A -85,B 0,C 180,E1 -11127.929,E2 -11127.929} C_VEL
LIN {X 0,Y 397.119,Z 139.021,A -85,B 0,C 180,E1 -11131.457,E2 -11131.457} C_VEL
LIN {X 0,Y 397.149,Z 139.01,A -85,B 0,C 180,E1 -11134.488,E2 -11134.488} C_VEL
LIN {X 0,Y 397.106,Z 139.02,A -85,B 0,C 180,E1 -11137.086,E2 -11137.086} C_VEL
LIN {X 0,Y 397.145,Z 139.011,A -85,B 0,C 180,E1 -11140.353,E2 -11140.353} C_VEL
LIN {X 0,Y 397.163,Z 139.012,A -85,B 0,C 180,E1 -11143.553,E2 -11143.553} C_VEL
LIN {X 0,Y 397.226,Z 139.003,A -85,B 0,C 180,E1 -11146.703,E2 -11146.703} C_VEL
LIN {X 0,Y 397.216,Z 139.003,A -85,B 0,C 180,E1 -11149.809,E2 -11149.809} C_VEL
LIN {X 0,Y 397.347,Z 138.991,A -85,B 0,C 180,E1 -11152.888,E2 -11152.888} C_VEL
LIN {X 0,Y 397.251,Z 139.004,A -85,B 0,C 180,E1 -11154.925,E2 -11154.925} C_VEL
LIN {X 0,Y 397.45,Z 138.973,A -85,B 0,C 180,E1 -11157.974,E2 -11157.974} C_VEL
LIN {X 0,Y 397.579,Z 138.957,A -85,B 0,C 180,E1 -11160,E2 -11160} C_VEL
LIN {X 0,Y 397.379,Z 138.986,A -85,B 0,C 180,E1 -11163.042,E2 -11163.042} C_VEL
LIN {X 0,Y 397.363,Z 138.987,A -85,B 0,C 180,E1 -11167.112,E2 -11167.112} C_VEL
LIN {X 0,Y 397.217,Z 139.004,A -85,B 0,C 180,E1 -11170.191,E2 -11170.191} C_VEL
LIN {X 0,Y 397.225,Z 139.002,A -85,B 0,C 180,E1 -11173.321,E2 -11173.321} C_VEL
LIN {X 0,Y 397.18,Z 139.007,A -85,B 0,C 180,E1 -11177.156,E2 -11177.156} C_VEL
LIN {X 0,Y 397.112,Z 139.019,A -85,B 0,C 180,E1 -11180.73,E2 -11180.73} C_VEL
LIN {X 0,Y 397.127,Z 139.016,A -85,B 0,C 180,E1 -11184.019,E2 -11184.019} C_VEL
LIN {X 0,Y 397.193,Z 139.005,A -85,B 0,C 180,E1 -11187.391,E2 -11187.391} C_VEL
LIN {X 0,Y 397.077,Z 139.02,A -85,B 0,C 180,E1 -11190.883,E2 -11190.883} C_VEL
LIN {X 0,Y 397.125,Z 139.016,A -85,B 0,C 180,E1 -11194.494,E2 -11194.494} C_VEL
LIN {X 0,Y 397.109,Z 139.02,A -85,B 0,C 180,E1 -11198.275,E2 -11198.275} C_VEL
LIN {X 0,Y 397.112,Z 139.015,A -85,B 0,C 180,E1 -11200.906,E2 -11200.906} C_VEL
LIN {X 0,Y 397.103,Z 139.02,A -85,B 0,C 180,E1 -11203.649,E2 -11203.649} C_VEL
LIN {X 0,Y 397.102,Z 139.017,A -85,B 0,C 180,E1 -11206.522,E2 -11206.522} C_VEL
LIN {X 0,Y 397.114,Z 139.016,A -85,B 0,C 180,E1 -11210.423,E2 -11210.423} C_VEL
LIN {X 0,Y 397.109,Z 139.017,A -85,B 0,C 180,E1 -11214.266,E2 -11214.266} C_VEL
LIN {X 0,Y 397.115,Z 139.015,A -85,B 0,C 180,E1 -11216.728,E2 -11216.728} C_VEL
LIN {X 0,Y 397.189,Z 139.092,A -85,B 0,C 180,E1 -11220.847,E2 -11220.847} C_VEL
LIN {X 0,Y 400.15,Z 153.609,A -85,B 0,C 180,E1 -11223.955,E2 -11223.955} C_VEL
LIN {X 0,Y 400.473,Z 157.843,A -85,B 0,C 180,E1 -11224.814,E2 -11224.814} C_VEL
LIN {X 0,Y 399.156,Z 175.839,A -85,B 0,C 180,E1 -11228.3,E2 -11228.3} C_VEL
LIN {X 0,Y 398.522,Z 186.434,A -85,B 0,C 180,E1 -11230.34,E2 -11230.34} C_VEL
LIN {X 0,Y 402.452,Z 216.934,A -85,B 0,C 180,E1 -11231.153,E2 -11231.153} C_VEL
LIN {X 0,Y 401.155,Z 295.562,A -85,B 0,C 180,E1 -11232.772,E2 -11232.772} C_VEL
LIN {X 0,Y 400.551,Z 308.926,A -85,B 0,C 180,E1 -11233.238,E2 -11233.238} C_VEL
LIN {X 0,Y 399.973,Z 321.288,A -85,B 0,C 180,E1 -11233.869,E2 -11233.869} C_VEL
LIN {X 0,Y 399.164,Z 333.22,A -85,B 0,C 180,E1 -11234.687,E2 -11234.687} C_VEL
LIN {X 0,Y 398.413,Z 344.741,A -85,B 0,C 180,E1 -11235.703,E2 -11235.703} C_VEL
LIN {X 0,Y 397.761,Z 355.17,A -85,B 0,C 180,E1 -11236.851,E2 -11236.851} C_VEL
LIN {X 0,Y 397.103,Z 365.357,A -85,B 0,C 180,E1 -11238.257,E2 -11238.257} C_VEL
LIN {X 0,Y 396.458,Z 374.307,A -85,B 0,C 180,E1 -11239.79,E2 -11239.79} C_VEL
LIN {X 0,Y 396.18,Z 381.44,A -85,B 0,C 180,E1 -11241.328,E2 -11241.328} C_VEL
LIN {X 0,Y 395.947,Z 387.118,A -85,B 0,C 180,E1 -11242.863,E2 -11242.863} C_VEL
LIN {X 0,Y 395.841,Z 391.012,A -85,B 0,C 180,E1 -11244.181,E2 -11244.181} C_VEL
LIN {X 0,Y 395.828,Z 394.849,A -85,B 0,C 180,E1 -11245.928,E2 -11245.928} C_VEL
LIN {X 0,Y 395.881,Z 396.477,A -85,B 0,C 180,E1 -11246.947,E2 -11246.947} C_VEL
LIN {X 0,Y 395.921,Z 397.673,A -85,B 0,C 180,E1 -11247.966,E2 -11247.966} C_VEL
LIN {X 0,Y 395.881,Z 398.394,A -85,B 0,C 180,E1 -11248.983,E2 -11248.983} C_VEL
LIN {X 0,Y 395.885,Z 398.702,A -85,B 0,C 180,E1 -11250,E2 -11250} C_VEL
LIN {X 0,Y 395.859,Z 398.599,A -85,B 0,C 180,E1 -11251.018,E2 -11251.018} C_VEL
LIN {X 0,Y 395.902,Z 398.08,A -85,B 0,C 180,E1 -11252.035,E2 -11252.035} C_VEL
LIN {X 0,Y 395.827,Z 397.097,A -85,B 0,C 180,E1 -11253.054,E2 -11253.054} C_VEL
LIN {X 0,Y 395.81,Z 395.701,A -85,B 0,C 180,E1 -11254.073,E2 -11254.073} C_VEL
LIN {X 0,Y 395.801,Z 392.414,A -85,B 0,C 180,E1 -11255.767,E2 -11255.767} C_VEL
LIN {X 0,Y 395.93,Z 388.793,A -85,B 0,C 180,E1 -11257.138,E2 -11257.138} C_VEL
LIN {X 0,Y 396.196,Z 383.649,A -85,B 0,C 180,E1 -11258.672,E2 -11258.672} C_VEL
LIN {X 0,Y 396.581,Z 377.196,A -85,B 0,C 180,E1 -11260.208,E2 -11260.208} C_VEL
LIN {X 0,Y 397.247,Z 369.176,A -85,B 0,C 180,E1 -11261.739,E2 -11261.739} C_VEL
LIN {X 0,Y 397.881,Z 361.011,A -85,B 0,C 180,E1 -11263.016,E2 -11263.016} C_VEL
LIN {X 0,Y 398.659,Z 351.094,A -85,B 0,C 180,E1 -11264.289,E2 -11264.289} C_VEL
LIN {X 0,Y 399.664,Z 340.132,A -85,B 0,C 180,E1 -11265.425,E2 -11265.425} C_VEL
LIN {X 0,Y 400.701,Z 327.761,A -85,B 0,C 180,E1 -11266.429,E2 -11266.429} C_VEL
LIN {X 0,Y 401.67,Z 314.717,A -85,B 0,C 180,E1 -11267.239,E2 -11267.239} C_VEL
LIN {X 0,Y 402.515,Z 301.353,A -85,B 0,C 180,E1 -11267.825,E2 -11267.825} C_VEL
LIN {X 0,Y 403.027,Z 287.204,A -85,B 0,C 180,E1 -11268.228,E2 -11268.228} C_VEL
LIN {X 0,Y 404.484,Z 216.788,A -85,B 0,C 180,E1 -11269.725,E2 -11269.725} C_VEL
LIN {X 0,Y 402.285,Z 199.904,A -85,B 0,C 180,E1 -11270.261,E2 -11270.261} C_VEL
LIN {X 0,Y 399.287,Z 183.292,A -85,B 0,C 180,E1 -11270.863,E2 -11270.863} C_VEL
LIN {X 0,Y 400.53,Z 166.211,A -85,B 0,C 180,E1 -11274.156,E2 -11274.156} C_VEL
LIN {X 0,Y 401.138,Z 156.958,A -85,B 0,C 180,E1 -11275.977,E2 -11275.977} C_VEL
LIN {X 0,Y 398.912,Z 146.068,A -85,B 0,C 180,E1 -11278.404,E2 -11278.404} C_VEL
LIN {X 0,Y 397.117,Z 139.027,A -85,B 0,C 180,E1 -11280.118,E2 -11280.118} C_VEL
LIN {X 0,Y 397.122,Z 139.02,A -85,B 0,C 180,E1 -11283.718,E2 -11283.718} C_VEL
LIN {X 0,Y 397.098,Z 139.02,A -85,B 0,C 180,E1 -11287.209,E2 -11287.209} C_VEL
LIN {X 0,Y 397.106,Z 139.021,A -85,B 0,C 180,E1 -11290.446,E2 -11290.446} C_VEL
LIN {X 0,Y 397.105,Z 139.021,A -85,B 0,C 180,E1 -11293.648,E2 -11293.648} C_VEL
LIN {X 0,Y 397.106,Z 139.017,A -85,B 0,C 180,E1 -11296.521,E2 -11296.521} C_VEL
LIN {X 0,Y 397.116,Z 139.012,A -85,B 0,C 180,E1 -11300.423,E2 -11300.423} C_VEL
LIN {X 0,Y 397.111,Z 139.015,A -85,B 0,C 180,E1 -11304.265,E2 -11304.265} C_VEL
LIN {X 0,Y 397.117,Z 139.013,A -85,B 0,C 180,E1 -11306.727,E2 -11306.727} C_VEL
LIN {X 0,Y 397.128,Z 139.015,A -85,B 0,C 180,E1 -11310.296,E2 -11310.296} C_VEL
LIN {X 0,Y 397.198,Z 139.007,A -85,B 0,C 180,E1 -11312.61,E2 -11312.61} C_VEL
LIN {X 0,Y 397.136,Z 139.014,A -85,B 0,C 180,E1 -11315.982,E2 -11315.982} C_VEL
LIN {X 0,Y 397.142,Z 139.012,A -85,B 0,C 180,E1 -11319.704,E2 -11319.704} C_VEL
LIN {X 0,Y 397.185,Z 139.008,A -85,B 0,C 180,E1 -11322.845,E2 -11322.845} C_VEL
LIN {X 0,Y 397.232,Z 139.003,A -85,B 0,C 180,E1 -11326.702,E2 -11326.702} C_VEL
LIN {X 0,Y 397.219,Z 139.006,A -85,B 0,C 180,E1 -11329.809,E2 -11329.809} C_VEL
LIN {X 0,Y 397.321,Z 138.997,A -85,B 0,C 180,E1 -11332.887,E2 -11332.887} C_VEL
LIN {X 0,Y 397.248,Z 139.008,A -85,B 0,C 180,E1 -11334.925,E2 -11334.925} C_VEL
LIN {X 0,Y 397.45,Z 138.981,A -85,B 0,C 180,E1 -11337.973,E2 -11337.973} C_VEL
LIN {X 0,Y 397.577,Z 138.963,A -85,B 0,C 180,E1 -11340,E2 -11340} C_VEL
LIN {X 0,Y 397.419,Z 139.012,A -85,B 0,C 180,E1 -11342.153,E2 -11342.153} C_VEL
LIN {X 0,Y 399.003,Z 146.946,A -85,B 0,C 180,E1 -11344.182,E2 -11344.182} C_VEL
LIN {X 0,Y 403.737,Z 158.278,A -85,B 0,C 180,E1 -11344.786,E2 -11344.786} C_VEL
LIN {X 0,Y 405.51,Z 166.131,A -85,B 0,C 180,E1 -11345.091,E2 -11345.091} C_VEL
LIN {X 0,Y 403.365,Z 254.272,A -85,B 0,C 180,E1 -11347.005,E2 -11347.005} C_VEL
LIN {X 0,Y 402.893,Z 268.152,A -85,B 0,C 180,E1 -11347.517,E2 -11347.517} C_VEL
LIN {X 0,Y 402.337,Z 280.176,A -85,B 0,C 180,E1 -11348.159,E2 -11348.159} C_VEL
LIN {X 0,Y 401.494,Z 292.808,A -85,B 0,C 180,E1 -11349.064,E2 -11349.064} C_VEL
LIN {X 0,Y 400.668,Z 304.077,A -85,B 0,C 180,E1 -11350.102,E2 -11350.102} C_VEL
LIN {X 0,Y 399.789,Z 314.232,A -85,B 0,C 180,E1 -11351.278,E2 -11351.278} C_VEL
LIN {X 0,Y 398.893,Z 324.256,A -85,B 0,C 180,E1 -11352.722,E2 -11352.722} C_VEL
LIN {X 0,Y 398.235,Z 331.028,A -85,B 0,C 180,E1 -11353.919,E2 -11353.919} C_VEL
LIN {X 0,Y 397.57,Z 337.842,A -85,B 0,C 180,E1 -11355.376,E2 -11355.376} C_VEL
LIN {X 0,Y 396.991,Z 344.056,A -85,B 0,C 180,E1 -11357.064,E2 -11357.064} C_VEL
LIN {X 0,Y 396.579,Z 348.433,A -85,B 0,C 180,E1 -11358.601,E2 -11358.601} C_VEL
LIN {X 0,Y 396.284,Z 351.398,A -85,B 0,C 180,E1 -11359.958,E2 -11359.958} C_VEL
LIN {X 0,Y 395.971,Z 354.188,A -85,B 0,C 180,E1 -11361.883,E2 -11361.883} C_VEL
LIN {X 0,Y 395.875,Z 355.135,A -85,B 0,C 180,E1 -11362.989,E2 -11362.989} C_VEL
LIN {X 0,Y 395.788,Z 355.561,A -85,B 0,C 180,E1 -11364.105,E2 -11364.105} C_VEL
LIN {X 0,Y 395.752,Z 355.501,A -85,B 0,C 180,E1 -11365.227,E2 -11365.227} C_VEL
LIN {X 0,Y 395.762,Z 354.954,A -85,B 0,C 180,E1 -11366.356,E2 -11366.356} C_VEL
LIN {X 0,Y 395.823,Z 353.846,A -85,B 0,C 180,E1 -11367.493,E2 -11367.493} C_VEL
LIN {X 0,Y 395.923,Z 352.243,A -85,B 0,C 180,E1 -11368.638,E2 -11368.638} C_VEL
LIN {X 0,Y 396.232,Z 348.708,A -85,B 0,C 180,E1 -11370.365,E2 -11370.365} C_VEL
LIN {X 0,Y 396.464,Z 343.682,A -85,B 0,C 180,E1 -11372.127,E2 -11372.127} C_VEL
LIN {X 0,Y 396.855,Z 337.993,A -85,B 0,C 180,E1 -11373.66,E2 -11373.66} C_VEL
LIN {X 0,Y 397.304,Z 331.391,A -85,B 0,C 180,E1 -11375.092,E2 -11375.092} C_VEL
LIN {X 0,Y 397.887,Z 322.81,A -85,B 0,C 180,E1 -11376.593,E2 -11376.593} C_VEL
LIN {X 0,Y 398.528,Z 313.488,A -85,B 0,C 180,E1 -11377.911,E2 -11377.911} C_VEL
LIN {X 0,Y 399.2,Z 302.663,A -85,B 0,C 180,E1 -11379.151,E2 -11379.151} C_VEL
LIN {X 0,Y 399.909,Z 290.682,A -85,B 0,C 180,E1 -11380.229,E2 -11380.229} C_VEL
LIN {X 0,Y 400.549,Z 278.43,A -85,B 0,C 180,E1 -11381.088,E2 -11381.088} C_VEL
LIN {X 0,Y 400.937,Z 265.335,A -85,B 0,C 180,E1 -11381.766,E2 -11381.766} C_VEL
LIN {X 0,Y 401.411,Z 251.983,A -85,B 0,C 180,E1 -11382.233,E2 -11382.233} C_VEL
LIN {X 0,Y 402.992,Z 164.356,A -85,B 0,C 180,E1 -11384.027,E2 -11384.027} C_VEL
LIN {X 0,Y 399.639,Z 149.137,A -85,B 0,C 180,E1 -11384.494,E2 -11384.494} C_VEL
LIN {X 0,Y 398.174,Z 144.291,A -85,B 0,C 180,E1 -11384.667,E2 -11384.667} C_VEL
LIN {X 0,Y 397.162,Z 139.015,A -85,B 0,C 180,E1 -11386.008,E2 -11386.008} C_VEL
LIN {X 0,Y 397.101,Z 139.022,A -85,B 0,C 180,E1 -11389.554,E2 -11389.554} C_VEL
LIN {X 0,Y 397.092,Z 139.018,A -85,B 0,C 180,E1 -11392.791,E2 -11392.791} C_VEL
LIN {X 0,Y 397.117,Z 139.015,A -85,B 0,C 180,E1 -11396.282,E2 -11396.282} C_VEL
LIN {X 0,Y 397.104,Z 139.017,A -85,B 0,C 180,E1 -11400.135,E2 -11400.135} C_VEL
LIN {X 0,Y 397.194,Z 139.005,A -85,B 0,C 180,E1 -11402.609,E2 -11402.609} C_VEL
LIN {X 0,Y 397.132,Z 139.013,A -85,B 0,C 180,E1 -11405.981,E2 -11405.981} C_VEL
LIN {X 0,Y 397.138,Z 139.014,A -85,B 0,C 180,E1 -11409.704,E2 -11409.704} C_VEL
LIN {X 0,Y 397.181,Z 139.01,A -85,B 0,C 180,E1 -11412.844,E2 -11412.844} C_VEL
LIN {X 0,Y 397.227,Z 139.003,A -85,B 0,C 180,E1 -11416.702,E2 -11416.702} C_VEL
LIN {X 0,Y 397.191,Z 139.007,A -85,B 0,C 180,E1 -11418.995,E2 -11418.995} C_VEL
LIN {X 0,Y 396.529,Z 139.088,A -85,B 0,C 180,E1 -11419.843,E2 -11419.843} C_VEL
LIN {X 0,Y 393.717,Z 139.442,A -85,B 0,C 180,E1 -11421.222,E2 -11421.222} C_VEL
LIN {X 0,Y 391.357,Z 139.735,A -85,B 0,C 180,E1 -11422.336,E2 -11422.336} C_VEL
LIN {X 0,Y 390.37,Z 139.859,A -85,B 0,C 180,E1 -11423.197,E2 -11423.197} C_VEL
LIN {X 0,Y 390.302,Z 139.863,A -85,B 0,C 180,E1 -11423.488,E2 -11423.488} C_VEL
LIN {X 0,Y 390.419,Z 139.849,A -85,B 0,C 180,E1 -11427.936,E2 -11427.936} C_VEL
LIN {X 0,Y 390.549,Z 139.833,A -85,B 0,C 180,E1 -11430,E2 -11430} C_VEL
LIN {X 0,Y 390.312,Z 139.865,A -85,B 0,C 180,E1 -11433.096,E2 -11433.096} C_VEL
LIN {X 0,Y 390.322,Z 139.863,A -85,B 0,C 180,E1 -11436.202,E2 -11436.202} C_VEL
LIN {X 0,Y 390.203,Z 139.876,A -85,B 0,C 180,E1 -11439.328,E2 -11439.328} C_VEL
LIN {X 0,Y 390.192,Z 139.877,A -85,B 0,C 180,E1 -11443.438,E2 -11443.438} C_VEL
LIN {X 0,Y 390.146,Z 139.883,A -85,B 0,C 180,E1 -11447.307,E2 -11447.307} C_VEL
LIN {X 0,Y 390.09,Z 139.896,A -85,B 0,C 180,E1 -11450.472,E2 -11450.472} C_VEL
LIN {X 0,Y 390.074,Z 139.896,A -85,B 0,C 180,E1 -11454.481,E2 -11454.481} C_VEL
LIN {X 0,Y 390.112,Z 139.892,A -85,B 0,C 180,E1 -11458.025,E2 -11458.025} C_VEL
LIN {X 0,Y 390.044,Z 139.897,A -85,B 0,C 180,E1 -11461.502,E2 -11461.502} C_VEL
LIN {X 0,Y 390.082,Z 139.891,A -85,B 0,C 180,E1 -11465.207,E2 -11465.207} C_VEL
LIN {X 0,Y 390.088,Z 139.89,A -85,B 0,C 180,E1 -11469.092,E2 -11469.092} C_VEL
LIN {X 0,Y 390.118,Z 139.888,A -85,B 0,C 180,E1 -11472.387,E2 -11472.387} C_VEL
LIN {X 0,Y 390.059,Z 139.896,A -85,B 0,C 180,E1 -11475.357,E2 -11475.357} C_VEL
LIN {X 0,Y 390.065,Z 139.895,A -85,B 0,C 180,E1 -11478.192,E2 -11478.192} C_VEL
LIN {X 0,Y 390.091,Z 139.89,A -85,B 0,C 180,E1 -11480.908,E2 -11480.908} C_VEL
LIN {X 0,Y 390.082,Z 139.891,A -85,B 0,C 180,E1 -11484.793,E2 -11484.793} C_VEL
LIN {X 0,Y 390.02,Z 139.899,A -85,B 0,C 180,E1 -11488.496,E2 -11488.496} C_VEL
LIN {X 0,Y 390.114,Z 139.888,A -85,B 0,C 180,E1 -11492.07,E2 -11492.07} C_VEL
LIN {X 0,Y 390.078,Z 139.897,A -85,B 0,C 180,E1 -11495.52,E2 -11495.52} C_VEL
LIN {X 0,Y 390.053,Z 139.897,A -85,B 0,C 180,E1 -11498.878,E2 -11498.878} C_VEL
LIN {X 0,Y 390.125,Z 139.886,A -85,B 0,C 180,E1 -11502.167,E2 -11502.167} C_VEL
LIN {X 0,Y 390.141,Z 139.888,A -85,B 0,C 180,E1 -11505.393,E2 -11505.393} C_VEL
LIN {X 0,Y 390.146,Z 139.884,A -85,B 0,C 180,E1 -11508.572,E2 -11508.572} C_VEL
LIN {X 0,Y 390.305,Z 139.863,A -85,B 0,C 180,E1 -11512.032,E2 -11512.032} C_VEL
LIN {X 0,Y 390.223,Z 139.878,A -85,B 0,C 180,E1 -11514.834,E2 -11514.834} C_VEL
LIN {X 0,Y 390.418,Z 139.849,A -85,B 0,C 180,E1 -11517.937,E2 -11517.937} C_VEL
LIN {X 0,Y 390.548,Z 139.833,A -85,B 0,C 180,E1 -11520,E2 -11520} C_VEL
LIN {X 0,Y 390.313,Z 139.866,A -85,B 0,C 180,E1 -11523.097,E2 -11523.097} C_VEL
LIN {X 0,Y 390.329,Z 139.862,A -85,B 0,C 180,E1 -11526.202,E2 -11526.202} C_VEL
LIN {X 0,Y 390.313,Z 139.865,A -85,B 0,C 180,E1 -11528.283,E2 -11528.283} C_VEL
LIN {X 0,Y 390.169,Z 139.885,A -85,B 0,C 180,E1 -11532.484,E2 -11532.484} C_VEL
LIN {X 0,Y 390.138,Z 139.884,A -85,B 0,C 180,E1 -11535.677,E2 -11535.677} C_VEL
LIN {X 0,Y 390.104,Z 139.89,A -85,B 0,C 180,E1 -11538.922,E2 -11538.922} C_VEL
LIN {X 0,Y 390.036,Z 139.902,A -85,B 0,C 180,E1 -11542.235,E2 -11542.235} C_VEL
LIN {X 0,Y 390.117,Z 139.888,A -85,B 0,C 180,E1 -11545.744,E2 -11545.744} C_VEL
LIN {X 0,Y 390.057,Z 139.894,A -85,B 0,C 180,E1 -11549.11,E2 -11549.11} C_VEL
LIN {X 0,Y 390.042,Z 139.897,A -85,B 0,C 180,E1 -11552.722,E2 -11552.722} C_VEL
LIN {X 0,Y 390.057,Z 139.898,A -85,B 0,C 180,E1 -11555.826,E2 -11555.826} C_VEL
LIN {X 0,Y 390.074,Z 139.892,A -85,B 0,C 180,E1 -11559.22,E2 -11559.22} C_VEL
LIN {X 0,Y 390.08,Z 139.893,A -85,B 0,C 180,E1 -11562.381,E2 -11562.381} C_VEL
LIN {X 0,Y 390.055,Z 139.898,A -85,B 0,C 180,E1 -11566.114,E2 -11566.114} C_VEL
LIN {X 0,Y 390.056,Z 139.898,A -85,B 0,C 180,E1 -11569.561,E2 -11569.561} C_VEL
LIN {X 0,Y 390.044,Z 139.896,A -85,B 0,C 180,E1 -11572.45,E2 -11572.45} C_VEL
LIN {X 0,Y 390.069,Z 139.896,A -85,B 0,C 180,E1 -11575.976,E2 -11575.976} C_VEL
LIN {X 0,Y 390.048,Z 139.899,A -85,B 0,C 180,E1 -11579.87,E2 -11579.87} C_VEL
LIN {X 0,Y 390.095,Z 139.93,A -85,B 0,C 180,E1 -11580.598,E2 -11580.598} C_VEL
LIN {X 0,Y 392.952,Z 153.748,A -85,B 0,C 180,E1 -11583.614,E2 -11583.614} C_VEL
LIN {X 0,Y 393.532,Z 158.563,A -85,B 0,C 180,E1 -11584.621,E2 -11584.621} C_VEL
LIN {X 0,Y 392.175,Z 176.502,A -85,B 0,C 180,E1 -11588.162,E2 -11588.162} C_VEL
LIN {X 0,Y 391.608,Z 186.036,A -85,B 0,C 180,E1 -11590.029,E2 -11590.029} C_VEL
LIN {X 0,Y 395.607,Z 217.466,A -85,B 0,C 180,E1 -11590.898,E2 -11590.898} C_VEL
LIN {X 0,Y 394.278,Z 295.041,A -85,B 0,C 180,E1 -11592.528,E2 -11592.528} C_VEL
LIN {X 0,Y 393.617,Z 309.164,A -85,B 0,C 180,E1 -11593.034,E2 -11593.034} C_VEL
LIN {X 0,Y 392.965,Z 321.85,A -85,B 0,C 180,E1 -11593.707,E2 -11593.707} C_VEL
LIN {X 0,Y 392.155,Z 333.562,A -85,B 0,C 180,E1 -11594.539,E2 -11594.539} C_VEL
LIN {X 0,Y 391.397,Z 344.686,A -85,B 0,C 180,E1 -11595.546,E2 -11595.546} C_VEL
LIN {X 0,Y 390.714,Z 355.256,A -85,B 0,C 180,E1 -11596.742,E2 -11596.742} C_VEL
LIN {X 0,Y 390.11,Z 364.534,A -85,B 0,C 180,E1 -11598.043,E2 -11598.043} C_VEL
LIN {X 0,Y 389.418,Z 373.563,A -85,B 0,C 180,E1 -11599.603,E2 -11599.603} C_VEL
LIN {X 0,Y 389.113,Z 380.789,A -85,B 0,C 180,E1 -11601.169,E2 -11601.169} C_VEL
LIN {X 0,Y 388.893,Z 386.526,A -85,B 0,C 180,E1 -11602.733,E2 -11602.733} C_VEL
LIN {X 0,Y 388.747,Z 390.836,A -85,B 0,C 180,E1 -11604.226,E2 -11604.226} C_VEL
LIN {X 0,Y 388.755,Z 394.352,A -85,B 0,C 180,E1 -11605.854,E2 -11605.854} C_VEL
LIN {X 0,Y 388.783,Z 395.999,A -85,B 0,C 180,E1 -11606.892,E2 -11606.892} C_VEL
LIN {X 0,Y 388.852,Z 397.222,A -85,B 0,C 180,E1 -11607.929,E2 -11607.929} C_VEL
LIN {X 0,Y 388.808,Z 397.972,A -85,B 0,C 180,E1 -11608.965,E2 -11608.965} C_VEL
LIN {X 0,Y 388.809,Z 398.296,A -85,B 0,C 180,E1 -11610,E2 -11610} C_VEL
LIN {X 0,Y 388.788,Z 398.211,A -85,B 0,C 180,E1 -11611.036,E2 -11611.036} C_VEL
LIN {X 0,Y 388.814,Z 397.716,A -85,B 0,C 180,E1 -11612.072,E2 -11612.072} C_VEL
LIN {X 0,Y 388.727,Z 396.754,A -85,B 0,C 180,E1 -11613.11,E2 -11613.11} C_VEL
LIN {X 0,Y 388.732,Z 395.376,A -85,B 0,C 180,E1 -11614.147,E2 -11614.147} C_VEL
LIN {X 0,Y 388.748,Z 393.575,A -85,B 0,C 180,E1 -11615.187,E2 -11615.187} C_VEL
LIN {X 0,Y 388.781,Z 389.979,A -85,B 0,C 180,E1 -11616.748,E2 -11616.748} C_VEL
LIN {X 0,Y 389.048,Z 385.276,A -85,B 0,C 180,E1 -11618.31,E2 -11618.31} C_VEL
LIN {X 0,Y 389.486,Z 378.178,A -85,B 0,C 180,E1 -11620.133,E2 -11620.133} C_VEL
LIN {X 0,Y 390.126,Z 370.492,A -85,B 0,C 180,E1 -11621.693,E2 -11621.693} C_VEL
LIN {X 0,Y 390.818,Z 362.688,A -85,B 0,C 180,E1 -11622.991,E2 -11622.991} C_VEL
LIN {X 0,Y 391.554,Z 353.626,A -85,B 0,C 180,E1 -11624.245,E2 -11624.245} C_VEL
LIN {X 0,Y 392.597,Z 342.889,A -85,B 0,C 180,E1 -11625.443,E2 -11625.443} C_VEL
LIN {X 0,Y 393.646,Z 331.444,A -85,B 0,C 180,E1 -11626.465,E2 -11626.465} C_VEL
LIN {X 0,Y 394.644,Z 319.682,A -85,B 0,C 180,E1 -11627.289,E2 -11627.289} C_VEL
LIN {X 0,Y 395.516,Z 307.069,A -85,B 0,C 180,E1 -11627.95,E2 -11627.95} C_VEL
LIN {X 0,Y 396.266,Z 293.219,A -85,B 0,C 180,E1 -11628.45,E2 -11628.45} C_VEL
LIN {X 0,Y 398.001,Z 217.828,A -85,B 0,C 180,E1 -11630.115,E2 -11630.115} C_VEL
LIN {X 0,Y 395.972,Z 201.928,A -85,B 0,C 180,E1 -11630.629,E2 -11630.629} C_VEL
LIN {X 0,Y 392.5,Z 182.775,A -85,B 0,C 180,E1 -11631.357,E2 -11631.357} C_VEL
LIN {X 0,Y 393.9,Z 165.275,A -85,B 0,C 180,E1 -11634.8,E2 -11634.8} C_VEL
LIN {X 0,Y 394.389,Z 159.829,A -85,B 0,C 180,E1 -11635.887,E2 -11635.887} C_VEL
LIN {X 0,Y 392.982,Z 151.706,A -85,B 0,C 180,E1 -11637.709,E2 -11637.709} C_VEL
LIN {X 0,Y 390.069,Z 139.915,A -85,B 0,C 180,E1 -11640.541,E2 -11640.541} C_VEL
LIN {X 0,Y 390.072,Z 139.898,A -85,B 0,C 180,E1 -11644.025,E2 -11644.025} C_VEL
LIN {X 0,Y 390.047,Z 139.9,A -85,B 0,C 180,E1 -11647.551,E2 -11647.551} C_VEL
LIN {X 0,Y 390.06,Z 139.898,A -85,B 0,C 180,E1 -11650.821,E2 -11650.821} C_VEL
LIN {X 0,Y 390.058,Z 139.897,A -85,B 0,C 180,E1 -11653.886,E2 -11653.886} C_VEL
LIN {X 0,Y 390.061,Z 139.894,A -85,B 0,C 180,E1 -11656.79,E2 -11656.79} C_VEL
LIN {X 0,Y 390.06,Z 139.896,A -85,B 0,C 180,E1 -11659.56,E2 -11659.56} C_VEL
LIN {X 0,Y 390.045,Z 139.894,A -85,B 0,C 180,E1 -11662.449,E2 -11662.449} C_VEL
LIN {X 0,Y 390.072,Z 139.89,A -85,B 0,C 180,E1 -11665.975,E2 -11665.975} C_VEL
LIN {X 0,Y 390.05,Z 139.899,A -85,B 0,C 180,E1 -11669.869,E2 -11669.869} C_VEL
LIN {X 0,Y 390.117,Z 139.892,A -85,B 0,C 180,E1 -11673.232,E2 -11673.232} C_VEL
LIN {X 0,Y 390.11,Z 139.889,A -85,B 0,C 180,E1 -11676.75,E2 -11676.75} C_VEL
LIN {X 0,Y 390.107,Z 139.888,A -85,B 0,C 180,E1 -11679.983,E2 -11679.983} C_VEL
LIN {X 0,Y 390.141,Z 139.888,A -85,B 0,C 180,E1 -11683.248,E2 -11683.248} C_VEL
LIN {X 0,Y 390.198,Z 139.879,A -85,B 0,C 180,E1 -11686.561,E2 -11686.561} C_VEL
LIN {X 0,Y 390.17,Z 139.884,A -85,B 0,C 180,E1 -11689.622,E2 -11689.622} C_VEL
LIN {X 0,Y 390.27,Z 139.874,A -85,B 0,C 180,E1 -11692.758,E2 -11692.758} C_VEL
LIN {X 0,Y 390.219,Z 139.884,A -85,B 0,C 180,E1 -11694.833,E2 -11694.833} C_VEL
LIN {X 0,Y 390.418,Z 139.857,A -85,B 0,C 180,E1 -11697.936,E2 -11697.936} C_VEL
LIN {X 0,Y 390.546,Z 139.839,A -85,B 0,C 180,E1 -11700,E2 -11700} C_VEL
LIN {X 0,Y 390.385,Z 139.907,A -85,B 0,C 180,E1 -11701.676,E2 -11701.676} C_VEL
LIN {X 0,Y 391.856,Z 147.358,A -85,B 0,C 180,E1 -11703.65,E2 -11703.65} C_VEL
LIN {X 0,Y 397.656,Z 161.027,A -85,B 0,C 180,E1 -11704.434,E2 -11704.434} C_VEL
LIN {X 0,Y 399.061,Z 168.045,A -85,B 0,C 180,E1 -11704.703,E2 -11704.703} C_VEL
LIN {X 0,Y 396.817,Z 254.926,A -85,B 0,C 180,E1 -11706.632,E2 -11706.632} C_VEL
LIN {X 0,Y 396.339,Z 268.163,A -85,B 0,C 180,E1 -11707.13,E2 -11707.13} C_VEL
LIN {X 0,Y 395.713,Z 280.289,A -85,B 0,C 180,E1 -11707.783,E2 -11707.783} C_VEL
LIN {X 0,Y 394.834,Z 292.938,A -85,B 0,C 180,E1 -11708.702,E2 -11708.702} C_VEL
LIN {X 0,Y 393.946,Z 304.23,A -85,B 0,C 180,E1 -11709.757,E2 -11709.757} C_VEL
LIN {X 0,Y 393.065,Z 313.987,A -85,B 0,C 180,E1 -11710.89,E2 -11710.89} C_VEL
LIN {X 0,Y 392.215,Z 322.853,A -85,B 0,C 180,E1 -11712.154,E2 -11712.154} C_VEL
LIN {X 0,Y 391.422,Z 330.6,A -85,B 0,C 180,E1 -11713.498,E2 -11713.498} C_VEL
LIN {X 0,Y 390.645,Z 338.173,A -85,B 0,C 180,E1 -11715.121,E2 -11715.121} C_VEL
LIN {X 0,Y 390.048,Z 344.159,A -85,B 0,C 180,E1 -11716.755,E2 -11716.755} C_VEL
LIN {X 0,Y 389.558,Z 348.805,A -85,B 0,C 180,E1 -11718.404,E2 -11718.404} C_VEL
LIN {X 0,Y 389.176,Z 352.322,A -85,B 0,C 180,E1 -11720.107,E2 -11720.107} C_VEL
LIN {X 0,Y 389.003,Z 353.931,A -85,B 0,C 180,E1 -11721.182,E2 -11721.182} C_VEL
LIN {X 0,Y 388.804,Z 355.471,A -85,B 0,C 180,E1 -11722.798,E2 -11722.798} C_VEL
LIN {X 0,Y 388.7,Z 356.016,A -85,B 0,C 180,E1 -11724.573,E2 -11724.573} C_VEL
LIN {X 0,Y 388.661,Z 355.693,A -85,B 0,C 180,E1 -11725.72,E2 -11725.72} C_VEL
LIN {X 0,Y 388.759,Z 354.039,A -85,B 0,C 180,E1 -11727.646,E2 -11727.646} C_VEL
LIN {X 0,Y 388.929,Z 351.626,A -85,B 0,C 180,E1 -11729.202,E2 -11729.202} C_VEL
LIN {X 0,Y 389.197,Z 347.657,A -85,B 0,C 180,E1 -11730.973,E2 -11730.973} C_VEL
LIN {X 0,Y 389.529,Z 342.098,A -85,B 0,C 180,E1 -11732.77,E2 -11732.77} C_VEL
LIN {X 0,Y 389.937,Z 336.251,A -85,B 0,C 180,E1 -11734.248,E2 -11734.248} C_VEL
LIN {X 0,Y 390.555,Z 327.954,A -85,B 0,C 180,E1 -11735.926,E2 -11735.926} C_VEL
LIN {X 0,Y 391.114,Z 319.236,A -85,B 0,C 180,E1 -11737.333,E2 -11737.333} C_VEL
LIN {X 0,Y 391.897,Z 308.551,A -85,B 0,C 180,E1 -11738.723,E2 -11738.723} C_VEL
LIN {X 0,Y 392.556,Z 298.257,A -85,B 0,C 180,E1 -11739.802,E2 -11739.802} C_VEL
LIN {X 0,Y 393.204,Z 286.138,A -85,B 0,C 180,E1 -11740.806,E2 -11740.806} C_VEL
LIN {X 0,Y 393.846,Z 273.75,A -85,B 0,C 180,E1 -11741.595,E2 -11741.595} C_VEL
LIN {X 0,Y 394.255,Z 260.892,A -85,B 0,C 180,E1 -11742.188,E2 -11742.188} C_VEL
LIN {X 0,Y 394.603,Z 247.289,A -85,B 0,C 180,E1 -11742.593,E2 -11742.593} C_VEL
LIN {X 0,Y 396.013,Z 164.691,A -85,B 0,C 180,E1 -11744.31,E2 -11744.31} C_VEL
LIN {X 0,Y 393.017,Z 151.075,A -85,B 0,C 180,E1 -11744.736,E2 -11744.736} C_VEL
LIN {X 0,Y 391.043,Z 144.577,A -85,B 0,C 180,E1 -11744.985,E2 -11744.985} C_VEL
LIN {X 0,Y 390.112,Z 139.893,A -85,B 0,C 180,E1 -11746.187,E2 -11746.187} C_VEL
LIN {X 0,Y 390.056,Z 139.9,A -85,B 0,C 180,E1 -11749.56,E2 -11749.56} C_VEL
LIN {X 0,Y 390.041,Z 139.896,A -85,B 0,C 180,E1 -11752.449,E2 -11752.449} C_VEL
LIN {X 0,Y 390.067,Z 139.895,A -85,B 0,C 180,E1 -11756.045,E2 -11756.045} C_VEL
LIN {X 0,Y 390.046,Z 139.898,A -85,B 0,C 180,E1 -11759.869,E2 -11759.869} C_VEL
LIN {X 0,Y 390.113,Z 139.892,A -85,B 0,C 180,E1 -11763.231,E2 -11763.231} C_VEL
LIN {X 0,Y 390.106,Z 139.889,A -85,B 0,C 180,E1 -11766.75,E2 -11766.75} C_VEL
LIN {X 0,Y 390.102,Z 139.889,A -85,B 0,C 180,E1 -11769.983,E2 -11769.983} C_VEL
LIN {X 0,Y 390.137,Z 139.89,A -85,B 0,C 180,E1 -11773.248,E2 -11773.248} C_VEL
LIN {X 0,Y 390.193,Z 139.879,A -85,B 0,C 180,E1 -11776.561,E2 -11776.561} C_VEL
LIN {X 0,Y 390.204,Z 139.879,A -85,B 0,C 180,E1 -11780.671,E2 -11780.671} C_VEL
LIN {X 0,Y 390.302,Z 139.863,A -85,B 0,C 180,E1 -11783.488,E2 -11783.488} C_VEL
LIN {X 0,Y 389.694,Z 139.942,A -85,B 0,C 180,E1 -11784.348,E2 -11784.348} C_VEL
LIN {X 0,Y 386.936,Z 140.283,A -85,B 0,C 180,E1 -11785.747,E2 -11785.747} C_VEL
LIN {X 0,Y 384.548,Z 140.587,A -85,B 0,C 180,E1 -11786.877,E2 -11786.877} C_VEL
LIN {X 0,Y 383.479,Z 140.714,A -85,B 0,C 180,E1 -11787.75,E2 -11787.75} C_VEL
LIN {X 0,Y 383.369,Z 140.727,A -85,B 0,C 180,E1 -11788.045,E2 -11788.045} C_VEL
LIN {X 0,Y 383.518,Z 140.709,A -85,B 0,C 180,E1 -11790,E2 -11790} C_VEL
LIN {X 0,Y 383.249,Z 140.745,A -85,B 0,C 180,E1 -11793.153,E2 -11793.153} C_VEL
LIN {X 0,Y 383.279,Z 140.741,A -85,B 0,C 180,E1 -11796.316,E2 -11796.316} C_VEL
LIN {X 0,Y 383.15,Z 140.755,A -85,B 0,C 180,E1 -11799.502,E2 -11799.502} C_VEL
LIN {X 0,Y 383.123,Z 140.758,A -85,B 0,C 180,E1 -11803.536,E2 -11803.536} C_VEL
LIN {X 0,Y 383.092,Z 140.762,A -85,B 0,C 180,E1 -11807.454,E2 -11807.454} C_VEL
LIN {X 0,Y 383.031,Z 140.773,A -85,B 0,C 180,E1 -11810.649,E2 -11810.649} C_VEL
LIN {X 0,Y 383.022,Z 140.772,A -85,B 0,C 180,E1 -11813.808,E2 -11813.808} C_VEL
LIN {X 0,Y 383.076,Z 140.769,A -85,B 0,C 180,E1 -11816.123,E2 -11816.123} C_VEL
LIN {X 0,Y 383.046,Z 140.771,A -85,B 0,C 180,E1 -11818.492,E2 -11818.492} C_VEL
LIN {X 0,Y 383.005,Z 140.776,A -85,B 0,C 180,E1 -11822.427,E2 -11822.427} C_VEL
LIN {X 0,Y 383.023,Z 140.776,A -85,B 0,C 180,E1 -11825.955,E2 -11825.955} C_VEL
LIN {X 0,Y 383.016,Z 140.774,A -85,B 0,C 180,E1 -11829.587,E2 -11829.587} C_VEL
LIN {X 0,Y 383.062,Z 140.766,A -85,B 0,C 180,E1 -11832.788,E2 -11832.788} C_VEL
LIN {X 0,Y 383.005,Z 140.779,A -85,B 0,C 180,E1 -11835.791,E2 -11835.791} C_VEL
LIN {X 0,Y 383.011,Z 140.772,A -85,B 0,C 180,E1 -11838.791,E2 -11838.791} C_VEL
LIN {X 0,Y 382.999,Z 140.776,A -85,B 0,C 180,E1 -11842.096,E2 -11842.096} C_VEL
LIN {X 0,Y 383.014,Z 140.775,A -85,B 0,C 180,E1 -11845.332,E2 -11845.332} C_VEL
LIN {X 0,Y 383.006,Z 140.776,A -85,B 0,C 180,E1 -11847.85,E2 -11847.85} C_VEL
LIN {X 0,Y 383.049,Z 140.771,A -85,B 0,C 180,E1 -11851.724,E2 -11851.724} C_VEL
LIN {X 0,Y 383.049,Z 140.77,A -85,B 0,C 180,E1 -11855.04,E2 -11855.04} C_VEL
LIN {X 0,Y 382.99,Z 140.774,A -85,B 0,C 180,E1 -11858.469,E2 -11858.469} C_VEL
LIN {X 0,Y 383.086,Z 140.764,A -85,B 0,C 180,E1 -11861.828,E2 -11861.828} C_VEL
LIN {X 0,Y 383.107,Z 140.766,A -85,B 0,C 180,E1 -11865.119,E2 -11865.119} C_VEL
LIN {X 0,Y 383.095,Z 140.762,A -85,B 0,C 180,E1 -11868.358,E2 -11868.358} C_VEL
LIN {X 0,Y 383.261,Z 140.741,A -85,B 0,C 180,E1 -11871.976,E2 -11871.976} C_VEL
LIN {X 0,Y 383.195,Z 140.753,A -85,B 0,C 180,E1 -11874.739,E2 -11874.739} C_VEL
LIN {X 0,Y 383.386,Z 140.725,A -85,B 0,C 180,E1 -11877.899,E2 -11877.899} C_VEL
LIN {X 0,Y 383.518,Z 140.709,A -85,B 0,C 180,E1 -11880,E2 -11880} C_VEL
LIN {X 0,Y 383.249,Z 140.745,A -85,B 0,C 180,E1 -11883.154,E2 -11883.154} C_VEL
LIN {X 0,Y 383.286,Z 140.74,A -85,B 0,C 180,E1 -11886.317,E2 -11886.317} C_VEL
LIN {X 0,Y 383.258,Z 140.745,A -85,B 0,C 180,E1 -11888.436,E2 -11888.436} C_VEL
LIN {X 0,Y 383.096,Z 140.761,A -85,B 0,C 180,E1 -11891.643,E2 -11891.643} C_VEL
LIN {X 0,Y 383.109,Z 140.763,A -85,B 0,C 180,E1 -11894.882,E2 -11894.882} C_VEL
LIN {X 0,Y 383.088,Z 140.765,A -85,B 0,C 180,E1 -11898.173,E2 -11898.173} C_VEL
LIN {X 0,Y 382.994,Z 140.774,A -85,B 0,C 180,E1 -11901.531,E2 -11901.531} C_VEL
LIN {X 0,Y 383.049,Z 140.768,A -85,B 0,C 180,E1 -11904.961,E2 -11904.961} C_VEL
LIN {X 0,Y 383.039,Z 140.772,A -85,B 0,C 180,E1 -11908.493,E2 -11908.493} C_VEL
LIN {X 0,Y 383.009,Z 140.779,A -85,B 0,C 180,E1 -11912.15,E2 -11912.15} C_VEL
LIN {X 0,Y 383.017,Z 140.772,A -85,B 0,C 180,E1 -11914.668,E2 -11914.668} C_VEL
LIN {X 0,Y 383.002,Z 140.778,A -85,B 0,C 180,E1 -11917.905,E2 -11917.905} C_VEL
LIN {X 0,Y 383.013,Z 140.772,A -85,B 0,C 180,E1 -11921.344,E2 -11921.344} C_VEL
LIN {X 0,Y 382.997,Z 140.776,A -85,B 0,C 180,E1 -11924.304,E2 -11924.304} C_VEL
LIN {X 0,Y 383.01,Z 140.773,A -85,B 0,C 180,E1 -11927.241,E2 -11927.241} C_VEL
LIN {X 0,Y 383.015,Z 140.772,A -85,B 0,C 180,E1 -11930.414,E2 -11930.414} C_VEL
LIN {X 0,Y 383.026,Z 140.773,A -85,B 0,C 180,E1 -11934.045,E2 -11934.045} C_VEL
LIN {X 0,Y 382.988,Z 140.781,A -85,B 0,C 180,E1 -11937.579,E2 -11937.579} C_VEL
LIN {X 0,Y 383.068,Z 140.961,A -85,B 0,C 180,E1 -11940.39,E2 -11940.39} C_VEL
LIN {X 0,Y 385.749,Z 153.649,A -85,B 0,C 180,E1 -11943.22,E2 -11943.22} C_VEL
LIN {X 0,Y 386.568,Z 159.245,A -85,B 0,C 180,E1 -11944.419,E2 -11944.419} C_VEL
LIN {X 0,Y 385.192,Z 177.243,A -85,B 0,C 180,E1 -11948.036,E2 -11948.036} C_VEL
LIN {X 0,Y 384.633,Z 185.763,A -85,B 0,C 180,E1 -11949.737,E2 -11949.737} C_VEL
LIN {X 0,Y 388.744,Z 218.743,A -85,B 0,C 180,E1 -11950.652,E2 -11950.652} C_VEL
LIN {X 0,Y 387.351,Z 295.343,A -85,B 0,C 180,E1 -11952.308,E2 -11952.308} C_VEL
LIN {X 0,Y 386.689,Z 309.231,A -85,B 0,C 180,E1 -11952.822,E2 -11952.822} C_VEL
LIN {X 0,Y 386.013,Z 321.26,A -85,B 0,C 180,E1 -11953.473,E2 -11953.473} C_VEL
LIN {X 0,Y 385.148,Z 333.811,A -85,B 0,C 180,E1 -11954.387,E2 -11954.387} C_VEL
LIN {X 0,Y 384.357,Z 344.881,A -85,B 0,C 180,E1 -11955.417,E2 -11955.417} C_VEL
LIN {X 0,Y 383.667,Z 355.277,A -85,B 0,C 180,E1 -11956.629,E2 -11956.629} C_VEL
LIN {X 0,Y 382.977,Z 365.326,A -85,B 0,C 180,E1 -11958.086,E2 -11958.086} C_VEL
LIN {X 0,Y 382.391,Z 372.78,A -85,B 0,C 180,E1 -11959.41,E2 -11959.41} C_VEL
LIN {X 0,Y 382.026,Z 380.107,A -85,B 0,C 180,E1 -11961.004,E2 -11961.004} C_VEL
LIN {X 0,Y 381.827,Z 385.912,A -85,B 0,C 180,E1 -11962.598,E2 -11962.598} C_VEL
LIN {X 0,Y 381.655,Z 390.636,A -85,B 0,C 180,E1 -11964.268,E2 -11964.268} C_VEL
LIN {X 0,Y 381.684,Z 393.842,A -85,B 0,C 180,E1 -11965.777,E2 -11965.777} C_VEL
LIN {X 0,Y 381.688,Z 395.509,A -85,B 0,C 180,E1 -11966.834,E2 -11966.834} C_VEL
LIN {X 0,Y 381.783,Z 396.756,A -85,B 0,C 180,E1 -11967.89,E2 -11967.89} C_VEL
LIN {X 0,Y 381.738,Z 397.547,A -85,B 0,C 180,E1 -11968.945,E2 -11968.945} C_VEL
LIN {X 0,Y 381.735,Z 397.89,A -85,B 0,C 180,E1 -11970,E2 -11970} C_VEL
LIN {X 0,Y 381.718,Z 397.821,A -85,B 0,C 180,E1 -11971.055,E2 -11971.055} C_VEL
LIN {X 0,Y 381.728,Z 397.347,A -85,B 0,C 180,E1 -11972.111,E2 -11972.111} C_VEL
LIN {X 0,Y 381.631,Z 396.416,A -85,B 0,C 180,E1 -11973.167,E2 -11973.167} C_VEL
LIN {X 0,Y 381.654,Z 395.055,A -85,B 0,C 180,E1 -11974.225,E2 -11974.225} C_VEL
LIN {X 0,Y 381.609,Z 391.783,A -85,B 0,C 180,E1 -11976.005,E2 -11976.005} C_VEL
LIN {X 0,Y 381.886,Z 386.749,A -85,B 0,C 180,E1 -11977.934,E2 -11977.934} C_VEL
LIN {X 0,Y 382.283,Z 380.203,A -85,B 0,C 180,E1 -11979.791,E2 -11979.791} C_VEL
LIN {X 0,Y 382.848,Z 373.122,A -85,B 0,C 180,E1 -11981.382,E2 -11981.382} C_VEL
LIN {X 0,Y 383.737,Z 364.329,A -85,B 0,C 180,E1 -11982.965,E2 -11982.965} C_VEL
LIN {X 0,Y 384.581,Z 354.405,A -85,B 0,C 180,E1 -11984.407,E2 -11984.407} C_VEL
LIN {X 0,Y 385.655,Z 344.344,A -85,B 0,C 180,E1 -11985.593,E2 -11985.593} C_VEL
LIN {X 0,Y 386.723,Z 333.408,A -85,B 0,C 180,E1 -11986.633,E2 -11986.633} C_VEL
LIN {X 0,Y 387.813,Z 321.299,A -85,B 0,C 180,E1 -11987.535,E2 -11987.535} C_VEL
LIN {X 0,Y 388.776,Z 308.879,A -85,B 0,C 180,E1 -11988.238,E2 -11988.238} C_VEL
LIN {X 0,Y 389.605,Z 296.137,A -85,B 0,C 180,E1 -11988.743,E2 -11988.743} C_VEL
LIN {X 0,Y 390.073,Z 277.937,A -85,B 0,C 180,E1 -11989.197,E2 -11989.197} C_VEL
LIN {X 0,Y 391.463,Z 218.101,A -85,B 0,C 180,E1 -11990.54,E2 -11990.54} C_VEL
LIN {X 0,Y 389.352,Z 201.483,A -85,B 0,C 180,E1 -11991.105,E2 -11991.105} C_VEL
LIN {X 0,Y 385.736,Z 182.287,A -85,B 0,C 180,E1 -11991.868,E2 -11991.868} C_VEL
LIN {X 0,Y 387.374,Z 164.131,A -85,B 0,C 180,E1 -11995.524,E2 -11995.524} C_VEL
LIN {X 0,Y 387.438,Z 160.043,A -85,B 0,C 180,E1 -11996.387,E2 -11996.387} C_VEL
LIN {X 0,Y 385.236,Z 149.461,A -85,B 0,C 180,E1 -11998.874,E2 -11998.874} C_VEL
LIN {X 0,Y 382.999,Z 140.783,A -85,B 0,C 180,E1 -12001.071,E2 -12001.071} C_VEL
LIN {X 0,Y 383.022,Z 140.777,A -85,B 0,C 180,E1 -12004.668,E2 -12004.668} C_VEL
LIN {X 0,Y 383.004,Z 140.78,A -85,B 0,C 180,E1 -12007.904,E2 -12007.904} C_VEL
LIN {X 0,Y 382.988,Z 140.78,A -85,B 0,C 180,E1 -12011.347,E2 -12011.347} C_VEL
LIN {X 0,Y 382.999,Z 140.776,A -85,B 0,C 180,E1 -12014.303,E2 -12014.303} C_VEL
LIN {X 0,Y 383.014,Z 140.773,A -85,B 0,C 180,E1 -12017.24,E2 -12017.24} C_VEL
LIN {X 0,Y 383.017,Z 140.769,A -85,B 0,C 180,E1 -12020.414,E2 -12020.414} C_VEL
LIN {X 0,Y 383.028,Z 140.77,A -85,B 0,C 180,E1 -12024.044,E2 -12024.044} C_VEL
LIN {X 0,Y 382.99,Z 140.777,A -85,B 0,C 180,E1 -12027.578,E2 -12027.578} C_VEL
LIN {X 0,Y 382.995,Z 140.776,A -85,B 0,C 180,E1 -12030.3,E2 -12030.3} C_VEL
LIN {X 0,Y 383.084,Z 140.76,A -85,B 0,C 180,E1 -12034.021,E2 -12034.021} C_VEL
LIN {X 0,Y 383.012,Z 140.773,A -85,B 0,C 180,E1 -12037.335,E2 -12037.335} C_VEL
LIN {X 0,Y 383.062,Z 140.769,A -85,B 0,C 180,E1 -12040.716,E2 -12040.716} C_VEL
LIN {X 0,Y 383.083,Z 140.764,A -85,B 0,C 180,E1 -12044.026,E2 -12044.026} C_VEL
LIN {X 0,Y 383.139,Z 140.761,A -85,B 0,C 180,E1 -12047.284,E2 -12047.284} C_VEL
LIN {X 0,Y 383.146,Z 140.759,A -85,B 0,C 180,E1 -12050.497,E2 -12050.497} C_VEL
LIN {X 0,Y 383.258,Z 140.748,A -85,B 0,C 180,E1 -12053.683,E2 -12053.683} C_VEL
LIN {X 0,Y 383.386,Z 140.733,A -85,B 0,C 180,E1 -12057.899,E2 -12057.899} C_VEL
LIN {X 0,Y 383.516,Z 140.715,A -85,B 0,C 180,E1 -12060,E2 -12060} C_VEL
LIN {X 0,Y 383.32,Z 140.858,A -85,B 0,C 180,E1 -12061.181,E2 -12061.181} C_VEL
LIN {X 0,Y 384.859,Z 147.896,A -85,B 0,C 180,E1 -12063.107,E2 -12063.107} C_VEL
LIN {X 0,Y 391.492,Z 163.27,A -85,B 0,C 180,E1 -12064.037,E2 -12064.037} C_VEL
LIN {X 0,Y 392.676,Z 169.365,A -85,B 0,C 180,E1 -12064.279,E2 -12064.279} C_VEL
LIN {X 0,Y 390.271,Z 255.371,A -85,B 0,C 180,E1 -12066.238,E2 -12066.238} C_VEL
LIN {X 0,Y 389.738,Z 269.051,A -85,B 0,C 180,E1 -12066.765,E2 -12066.765} C_VEL
LIN {X 0,Y 389.069,Z 281.504,A -85,B 0,C 180,E1 -12067.46,E2 -12067.46} C_VEL
LIN {X 0,Y 388.201,Z 293.202,A -85,B 0,C 180,E1 -12068.327,E2 -12068.327} C_VEL
LIN {X 0,Y 387.257,Z 304.534,A -85,B 0,C 180,E1 -12069.4,E2 -12069.4} C_VEL
LIN {X 0,Y 386.218,Z 315.322,A -85,B 0,C 180,E1 -12070.691,E2 -12070.691} C_VEL
LIN {X 0,Y 385.228,Z 324.83,A -85,B 0,C 180,E1 -12072.11,E2 -12072.11} C_VEL
LIN {X 0,Y 384.401,Z 332.311,A -85,B 0,C 180,E1 -12073.48,E2 -12073.48} C_VEL
LIN {X 0,Y 383.591,Z 339.607,A -85,B 0,C 180,E1 -12075.134,E2 -12075.134} C_VEL
LIN {X 0,Y 383.069,Z 344.523,A -85,B 0,C 180,E1 -12076.521,E2 -12076.521} C_VEL
LIN {X 0,Y 382.553,Z 349.181,A -85,B 0,C 180,E1 -12078.198,E2 -12078.198} C_VEL
LIN {X 0,Y 382.284,Z 351.615,A -85,B 0,C 180,E1 -12079.324,E2 -12079.324} C_VEL
LIN {X 0,Y 382.035,Z 353.564,A -85,B 0,C 180,E1 -12080.458,E2 -12080.458} C_VEL
LIN {X 0,Y 381.877,Z 354.966,A -85,B 0,C 180,E1 -12081.597,E2 -12081.597} C_VEL
LIN {X 0,Y 381.706,Z 356.059,A -85,B 0,C 180,E1 -12082.985,E2 -12082.985} C_VEL
LIN {X 0,Y 381.611,Z 356.313,A -85,B 0,C 180,E1 -12085.061,E2 -12085.061} C_VEL
LIN {X 0,Y 381.598,Z 355.781,A -85,B 0,C 180,E1 -12086.232,E2 -12086.232} C_VEL
LIN {X 0,Y 381.682,Z 354.116,A -85,B 0,C 180,E1 -12087.891,E2 -12087.891} C_VEL
LIN {X 0,Y 381.931,Z 350.875,A -85,B 0,C 180,E1 -12089.79,E2 -12089.79} C_VEL
LIN {X 0,Y 382.191,Z 346.4,A -85,B 0,C 180,E1 -12091.606,E2 -12091.606} C_VEL
LIN {X 0,Y 382.623,Z 340.319,A -85,B 0,C 180,E1 -12093.438,E2 -12093.438} C_VEL
LIN {X 0,Y 383.06,Z 333.75,A -85,B 0,C 180,E1 -12094.983,E2 -12094.983} C_VEL
LIN {X 0,Y 383.678,Z 326.259,A -85,B 0,C 180,E1 -12096.414,E2 -12096.414} C_VEL
LIN {X 0,Y 384.283,Z 317.542,A -85,B 0,C 180,E1 -12097.782,E2 -12097.782} C_VEL
LIN {X 0,Y 384.994,Z 307.764,A -85,B 0,C 180,E1 -12099.034,E2 -12099.034} C_VEL
LIN {X 0,Y 385.733,Z 296.794,A -85,B 0,C 180,E1 -12100.161,E2 -12100.161} C_VEL
LIN {X 0,Y 386.422,Z 284.572,A -85,B 0,C 180,E1 -12101.158,E2 -12101.158} C_VEL
LIN {X 0,Y 387.034,Z 272.055,A -85,B 0,C 180,E1 -12101.927,E2 -12101.927} C_VEL
LIN {X 0,Y 387.376,Z 259.366,A -85,B 0,C 180,E1 -12102.495,E2 -12102.495} C_VEL
LIN {X 0,Y 387.781,Z 245.6,A -85,B 0,C 180,E1 -12102.881,E2 -12102.881} C_VEL
LIN {X 0,Y 389.259,Z 165.814,A -85,B 0,C 180,E1 -12104.574,E2 -12104.574} C_VEL
LIN {X 0,Y 386.392,Z 153.031,A -85,B 0,C 180,E1 -12104.985,E2 -12104.985} C_VEL
LIN {X 0,Y 383.872,Z 144.985,A -85,B 0,C 180,E1 -12105.287,E2 -12105.287} C_VEL
LIN {X 0,Y 383.081,Z 140.768,A -85,B 0,C 180,E1 -12106.394,E2 -12106.394} C_VEL
LIN {X 0,Y 383.013,Z 140.772,A -85,B 0,C 180,E1 -12110.413,E2 -12110.413} C_VEL
LIN {X 0,Y 383.024,Z 140.772,A -85,B 0,C 180,E1 -12114.044,E2 -12114.044} C_VEL
LIN {X 0,Y 382.986,Z 140.781,A -85,B 0,C 180,E1 -12117.578,E2 -12117.578} C_VEL
LIN {X 0,Y 382.991,Z 140.774,A -85,B 0,C 180,E1 -12120.3,E2 -12120.3} C_VEL
LIN {X 0,Y 383.056,Z 140.767,A -85,B 0,C 180,E1 -12122.698,E2 -12122.698} C_VEL
LIN {X 0,Y 383.033,Z 140.769,A -85,B 0,C 180,E1 -12126.192,E2 -12126.192} C_VEL
LIN {X 0,Y 383.054,Z 140.769,A -85,B 0,C 180,E1 -12129.598,E2 -12129.598} C_VEL
LIN {X 0,Y 383.093,Z 140.766,A -85,B 0,C 180,E1 -12132.93,E2 -12132.93} C_VEL
LIN {X 0,Y 383.124,Z 140.759,A -85,B 0,C 180,E1 -12136.463,E2 -12136.463} C_VEL
LIN {X 0,Y 383.151,Z 140.756,A -85,B 0,C 180,E1 -12140.498,E2 -12140.498} C_VEL
LIN {X 0,Y 383.279,Z 140.739,A -85,B 0,C 180,E1 -12143.683,E2 -12143.683} C_VEL
LIN {X 0,Y 383.369,Z 140.727,A -85,B 0,C 180,E1 -12148.045,E2 -12148.045} C_VEL
LIN {X 0,Y 382.659,Z 140.821,A -85,B 0,C 180,E1 -12148.922,E2 -12148.922} C_VEL
LIN {X 0,Y 379.844,Z 141.168,A -85,B 0,C 180,E1 -12150.349,E2 -12150.349} C_VEL
LIN {X 0,Y 377.453,Z 141.465,A -85,B 0,C 180,E1 -12151.502,E2 -12151.502} C_VEL
LIN {X 0,Y 376.37,Z 141.602,A -85,B 0,C 180,E1 -12152.392,E2 -12152.392} C_VEL
LIN {X 0,Y 376.25,Z 141.613,A -85,B 0,C 180,E1 -12152.694,E2 -12152.694} C_VEL
LIN {X 0,Y 376.237,Z 141.62,A -85,B 0,C 180,E1 -12156.435,E2 -12156.435} C_VEL
LIN {X 0,Y 376.117,Z 141.631,A -85,B 0,C 180,E1 -12159.681,E2 -12159.681} C_VEL
LIN {X 0,Y 376.087,Z 141.634,A -85,B 0,C 180,E1 -12163.657,E2 -12163.657} C_VEL
LIN {X 0,Y 376.042,Z 141.64,A -85,B 0,C 180,E1 -12167.607,E2 -12167.607} C_VEL
LIN {X 0,Y 375.975,Z 141.65,A -85,B 0,C 180,E1 -12170.832,E2 -12170.832} C_VEL
LIN {X 0,Y 375.986,Z 141.654,A -85,B 0,C 180,E1 -12174.281,E2 -12174.281} C_VEL
LIN {X 0,Y 376.016,Z 141.645,A -85,B 0,C 180,E1 -12176.652,E2 -12176.652} C_VEL
LIN {X 0,Y 375.973,Z 141.649,A -85,B 0,C 180,E1 -12179.078,E2 -12179.078} C_VEL
LIN {X 0,Y 375.955,Z 141.651,A -85,B 0,C 180,E1 -12182.827,E2 -12182.827} C_VEL
LIN {X 0,Y 375.955,Z 141.652,A -85,B 0,C 180,E1 -12185.415,E2 -12185.415} C_VEL
LIN {X 0,Y 375.972,Z 141.652,A -85,B 0,C 180,E1 -12188.271,E2 -12188.271} C_VEL
LIN {X 0,Y 375.985,Z 141.65,A -85,B 0,C 180,E1 -12191.61,E2 -12191.61} C_VEL
LIN {X 0,Y 375.967,Z 141.651,A -85,B 0,C 180,E1 -12195.262,E2 -12195.262} C_VEL
LIN {X 0,Y 375.977,Z 141.649,A -85,B 0,C 180,E1 -12199.138,E2 -12199.138} C_VEL
LIN {X 0,Y 375.964,Z 141.654,A -85,B 0,C 180,E1 -12201.912,E2 -12201.912} C_VEL
LIN {X 0,Y 375.976,Z 141.652,A -85,B 0,C 180,E1 -12205.333,E2 -12205.333} C_VEL
LIN {X 0,Y 375.954,Z 141.651,A -85,B 0,C 180,E1 -12208.438,E2 -12208.438} C_VEL
LIN {X 0,Y 375.992,Z 141.647,A -85,B 0,C 180,E1 -12212.142,E2 -12212.142} C_VEL
LIN {X 0,Y 376.003,Z 141.645,A -85,B 0,C 180,E1 -12214.539,E2 -12214.539} C_VEL
LIN {X 0,Y 375.96,Z 141.651,A -85,B 0,C 180,E1 -12218.046,E2 -12218.046} C_VEL
LIN {X 0,Y 376.021,Z 141.647,A -85,B 0,C 180,E1 -12221.474,E2 -12221.474} C_VEL
LIN {X 0,Y 376.055,Z 141.641,A -85,B 0,C 180,E1 -12224.833,E2 -12224.833} C_VEL
LIN {X 0,Y 376.047,Z 141.639,A -85,B 0,C 180,E1 -12228.137,E2 -12228.137} C_VEL
LIN {X 0,Y 376.216,Z 141.618,A -85,B 0,C 180,E1 -12231.919,E2 -12231.919} C_VEL
LIN {X 0,Y 376.167,Z 141.627,A -85,B 0,C 180,E1 -12234.64,E2 -12234.64} C_VEL
LIN {X 0,Y 376.352,Z 141.601,A -85,B 0,C 180,E1 -12237.86,E2 -12237.86} C_VEL
LIN {X 0,Y 376.487,Z 141.585,A -85,B 0,C 180,E1 -12240,E2 -12240} C_VEL
LIN {X 0,Y 376.187,Z 141.624,A -85,B 0,C 180,E1 -12243.213,E2 -12243.213} C_VEL
LIN {X 0,Y 376.246,Z 141.618,A -85,B 0,C 180,E1 -12246.435,E2 -12246.435} C_VEL
LIN {X 0,Y 376.204,Z 141.625,A -85,B 0,C 180,E1 -12248.596,E2 -12248.596} C_VEL
LIN {X 0,Y 376.048,Z 141.64,A -85,B 0,C 180,E1 -12251.864,E2 -12251.864} C_VEL
LIN {X 0,Y 376.057,Z 141.639,A -85,B 0,C 180,E1 -12255.168,E2 -12255.168} C_VEL
LIN {X 0,Y 376.023,Z 141.648,A -85,B 0,C 180,E1 -12258.526,E2 -12258.526} C_VEL
LIN {X 0,Y 375.957,Z 141.653,A -85,B 0,C 180,E1 -12261.955,E2 -12261.955} C_VEL
LIN {X 0,Y 376.004,Z 141.645,A -85,B 0,C 180,E1 -12265.462,E2 -12265.462} C_VEL
LIN {X 0,Y 375.969,Z 141.649,A -85,B 0,C 180,E1 -12269.08,E2 -12269.08} C_VEL
LIN {X 0,Y 375.95,Z 141.652,A -85,B 0,C 180,E1 -12272.829,E2 -12272.829} C_VEL
LIN {X 0,Y 375.958,Z 141.651,A -85,B 0,C 180,E1 -12275.416,E2 -12275.416} C_VEL
LIN {X 0,Y 375.977,Z 141.652,A -85,B 0,C 180,E1 -12278.272,E2 -12278.272} C_VEL
LIN {X 0,Y 375.96,Z 141.653,A -85,B 0,C 180,E1 -12281.606,E2 -12281.606} C_VEL
LIN {X 0,Y 375.927,Z 141.655,A -85,B 0,C 180,E1 -12285.269,E2 -12285.269} C_VEL
LIN {X 0,Y 375.934,Z 141.655,A -85,B 0,C 180,E1 -12288.4,E2 -12288.4} C_VEL
LIN {X 0,Y 375.974,Z 141.655,A -85,B 0,C 180,E1 -12291.73,E2 -12291.73} C_VEL
LIN {X 0,Y 375.981,Z 141.65,A -85,B 0,C 180,E1 -12295.333,E2 -12295.333} C_VEL
LIN {X 0,Y 375.959,Z 141.653,A -85,B 0,C 180,E1 -12298.439,E2 -12298.439} C_VEL
LIN {X 0,Y 375.994,Z 141.719,A -85,B 0,C 180,E1 -12300.116,E2 -12300.116} C_VEL
LIN {X 0,Y 378.825,Z 155.068,A -85,B 0,C 180,E1 -12303.149,E2 -12303.149} C_VEL
LIN {X 0,Y 379.561,Z 159.902,A -85,B 0,C 180,E1 -12304.207,E2 -12304.207} C_VEL
LIN {X 0,Y 378.617,Z 172.367,A -85,B 0,C 180,E1 -12306.769,E2 -12306.769} C_VEL
LIN {X 0,Y 377.692,Z 185.349,A -85,B 0,C 180,E1 -12309.409,E2 -12309.409} C_VEL
LIN {X 0,Y 381.889,Z 219.991,A -85,B 0,C 180,E1 -12310.403,E2 -12310.403} C_VEL
LIN {X 0,Y 380.488,Z 294.509,A -85,B 0,C 180,E1 -12312.048,E2 -12312.048} C_VEL
LIN {X 0,Y 379.82,Z 308.513,A -85,B 0,C 180,E1 -12312.571,E2 -12312.571} C_VEL
LIN {X 0,Y 379.095,Z 320.631,A -85,B 0,C 180,E1 -12313.232,E2 -12313.232} C_VEL
LIN {X 0,Y 378.241,Z 332.438,A -85,B 0,C 180,E1 -12314.094,E2 -12314.094} C_VEL
LIN {X 0,Y 377.469,Z 343.913,A -85,B 0,C 180,E1 -12315.167,E2 -12315.167} C_VEL
LIN {X 0,Y 376.694,Z 354.281,A -85,B 0,C 180,E1 -12316.377,E2 -12316.377} C_VEL
LIN {X 0,Y 375.99,Z 364.44,A -85,B 0,C 180,E1 -12317.861,E2 -12317.861} C_VEL
LIN {X 0,Y 375.272,Z 373.358,A -85,B 0,C 180,E1 -12319.479,E2 -12319.479} C_VEL
LIN {X 0,Y 374.948,Z 380.459,A -85,B 0,C 180,E1 -12321.105,E2 -12321.105} C_VEL
LIN {X 0,Y 374.67,Z 386.941,A -85,B 0,C 180,E1 -12322.997,E2 -12322.997} C_VEL
LIN {X 0,Y 374.597,Z 391.148,A -85,B 0,C 180,E1 -12324.618,E2 -12324.618} C_VEL
LIN {X 0,Y 374.616,Z 393.325,A -85,B 0,C 180,E1 -12325.697,E2 -12325.697} C_VEL
LIN {X 0,Y 374.595,Z 395.014,A -85,B 0,C 180,E1 -12326.774,E2 -12326.774} C_VEL
LIN {X 0,Y 374.715,Z 396.285,A -85,B 0,C 180,E1 -12327.851,E2 -12327.851} C_VEL
LIN {X 0,Y 374.67,Z 397.115,A -85,B 0,C 180,E1 -12328.926,E2 -12328.926} C_VEL
LIN {X 0,Y 374.664,Z 397.482,A -85,B 0,C 180,E1 -12330,E2 -12330} C_VEL
LIN {X 0,Y 374.65,Z 397.433,A -85,B 0,C 180,E1 -12331.075,E2 -12331.075} C_VEL
LIN {X 0,Y 374.628,Z 396.976,A -85,B 0,C 180,E1 -12332.151,E2 -12332.151} C_VEL
LIN {X 0,Y 374.54,Z 396.085,A -85,B 0,C 180,E1 -12333.227,E2 -12333.227} C_VEL
LIN {X 0,Y 374.576,Z 394.741,A -85,B 0,C 180,E1 -12334.304,E2 -12334.304} C_VEL
LIN {X 0,Y 374.513,Z 391.837,A -85,B 0,C 180,E1 -12335.963,E2 -12335.963} C_VEL
LIN {X 0,Y 374.723,Z 388.05,A -85,B 0,C 180,E1 -12337.544,E2 -12337.544} C_VEL
LIN {X 0,Y 375.02,Z 383.028,A -85,B 0,C 180,E1 -12339.166,E2 -12339.166} C_VEL
LIN {X 0,Y 375.489,Z 376.712,A -85,B 0,C 180,E1 -12340.788,E2 -12340.788} C_VEL
LIN {X 0,Y 376.345,Z 368.916,A -85,B 0,C 180,E1 -12342.402,E2 -12342.402} C_VEL
LIN {X 0,Y 377.056,Z 360.995,A -85,B 0,C 180,E1 -12343.748,E2 -12343.748} C_VEL
LIN {X 0,Y 378.045,Z 351.383,A -85,B 0,C 180,E1 -12345.086,E2 -12345.086} C_VEL
LIN {X 0,Y 379.323,Z 339.478,A -85,B 0,C 180,E1 -12346.413,E2 -12346.413} C_VEL
LIN {X 0,Y 380.596,Z 327.384,A -85,B 0,C 180,E1 -12347.462,E2 -12347.462} C_VEL
LIN {X 0,Y 381.634,Z 314.662,A -85,B 0,C 180,E1 -12348.314,E2 -12348.314} C_VEL
LIN {X 0,Y 382.711,Z 301.252,A -85,B 0,C 180,E1 -12348.954,E2 -12348.954} C_VEL
LIN {X 0,Y 383.293,Z 288.072,A -85,B 0,C 180,E1 -12349.376,E2 -12349.376} C_VEL
LIN {X 0,Y 385.085,Z 219.119,A -85,B 0,C 180,E1 -12350.966,E2 -12350.966} C_VEL
LIN {X 0,Y 383.023,Z 202.874,A -85,B 0,C 180,E1 -12351.538,E2 -12351.538} C_VEL
LIN {X 0,Y 379.45,Z 184.064,A -85,B 0,C 180,E1 -12352.312,E2 -12352.312} C_VEL
LIN {X 0,Y 379.007,Z 181.607,A -85,B 0,C 180,E1 -12352.452,E2 -12352.452} C_VEL
LIN {X 0,Y 380.578,Z 165.702,A -85,B 0,C 180,E1 -12355.72,E2 -12355.72} C_VEL
LIN {X 0,Y 380.645,Z 161.756,A -85,B 0,C 180,E1 -12356.57,E2 -12356.57} C_VEL
LIN {X 0,Y 378.702,Z 152.303,A -85,B 0,C 180,E1 -12358.85,E2 -12358.85} C_VEL
LIN {X 0,Y 375.953,Z 141.661,A -85,B 0,C 180,E1 -12361.641,E2 -12361.641} C_VEL
LIN {X 0,Y 375.961,Z 141.654,A -85,B 0,C 180,E1 -12365.416,E2 -12365.416} C_VEL
LIN {X 0,Y 375.978,Z 141.653,A -85,B 0,C 180,E1 -12368.271,E2 -12368.271} C_VEL
LIN {X 0,Y 375.938,Z 141.658,A -85,B 0,C 180,E1 -12371.601,E2 -12371.601} C_VEL
LIN {X 0,Y 375.93,Z 141.658,A -85,B 0,C 180,E1 -12375.269,E2 -12375.269} C_VEL
LIN {X 0,Y 375.938,Z 141.65,A -85,B 0,C 180,E1 -12378.399,E2 -12378.399} C_VEL
LIN {X 0,Y 375.976,Z 141.648,A -85,B 0,C 180,E1 -12381.73,E2 -12381.73} C_VEL
LIN {X 0,Y 375.983,Z 141.647,A -85,B 0,C 180,E1 -12385.333,E2 -12385.333} C_VEL
LIN {X 0,Y 375.961,Z 141.647,A -85,B 0,C 180,E1 -12388.438,E2 -12388.438} C_VEL
LIN {X 0,Y 375.987,Z 141.649,A -85,B 0,C 180,E1 -12392.14,E2 -12392.14} C_VEL
LIN {X 0,Y 376.01,Z 141.641,A -85,B 0,C 180,E1 -12394.539,E2 -12394.539} C_VEL
LIN {X 0,Y 375.967,Z 141.652,A -85,B 0,C 180,E1 -12398.046,E2 -12398.046} C_VEL
LIN {X 0,Y 376.006,Z 141.644,A -85,B 0,C 180,E1 -12401.473,E2 -12401.473} C_VEL
LIN {X 0,Y 376.061,Z 141.639,A -85,B 0,C 180,E1 -12404.832,E2 -12404.832} C_VEL
LIN {X 0,Y 376.052,Z 141.643,A -85,B 0,C 180,E1 -12408.136,E2 -12408.136} C_VEL
LIN {X 0,Y 376.196,Z 141.627,A -85,B 0,C 180,E1 -12411.946,E2 -12411.946} C_VEL
LIN {X 0,Y 376.162,Z 141.634,A -85,B 0,C 180,E1 -12414.639,E2 -12414.639} C_VEL
LIN {X 0,Y 376.352,Z 141.61,A -85,B 0,C 180,E1 -12417.859,E2 -12417.859} C_VEL
LIN {X 0,Y 376.352,Z 141.607,A -85,B 0,C 180,E1 -12420.535,E2 -12420.535} C_VEL
LIN {X 0,Y 377.872,Z 148.483,A -85,B 0,C 180,E1 -12422.551,E2 -12422.551} C_VEL
LIN {X 0,Y 385.484,Z 166.091,A -85,B 0,C 180,E1 -12423.652,E2 -12423.652} C_VEL
LIN {X 0,Y 386.315,Z 169.876,A -85,B 0,C 180,E1 -12423.813,E2 -12423.813} C_VEL
LIN {X 0,Y 383.788,Z 255.473,A -85,B 0,C 180,E1 -12425.813,E2 -12425.813} C_VEL
LIN {X 0,Y 383.21,Z 269.249,A -85,B 0,C 180,E1 -12426.352,E2 -12426.352} C_VEL
LIN {X 0,Y 382.449,Z 282.377,A -85,B 0,C 180,E1 -12427.103,E2 -12427.103} C_VEL
LIN {X 0,Y 381.47,Z 295.036,A -85,B 0,C 180,E1 -12428.075,E2 -12428.075} C_VEL
LIN {X 0,Y 380.454,Z 306.111,A -85,B 0,C 180,E1 -12429.167,E2 -12429.167} C_VEL
LIN {X 0,Y 379.445,Z 316.1,A -85,B 0,C 180,E1 -12430.404,E2 -12430.404} C_VEL
LIN {X 0,Y 378.436,Z 325.201,A -85,B 0,C 180,E1 -12431.787,E2 -12431.787} C_VEL
LIN {X 0,Y 377.558,Z 332.692,A -85,B 0,C 180,E1 -12433.18,E2 -12433.18} C_VEL
LIN {X 0,Y 376.67,Z 340.018,A -85,B 0,C 180,E1 -12434.874,E2 -12434.874} C_VEL
LIN {X 0,Y 376.102,Z 344.899,A -85,B 0,C 180,E1 -12436.277,E2 -12436.277} C_VEL
LIN {X 0,Y 375.549,Z 349.557,A -85,B 0,C 180,E1 -12437.985,E2 -12437.985} C_VEL
LIN {X 0,Y 375.121,Z 353.03,A -85,B 0,C 180,E1 -12439.708,E2 -12439.708} C_VEL
LIN {X 0,Y 374.896,Z 354.718,A -85,B 0,C 180,E1 -12440.866,E2 -12440.866} C_VEL
LIN {X 0,Y 374.726,Z 355.915,A -85,B 0,C 180,E1 -12442.03,E2 -12442.03} C_VEL
LIN {X 0,Y 374.605,Z 356.598,A -85,B 0,C 180,E1 -12443.202,E2 -12443.202} C_VEL
LIN {X 0,Y 374.537,Z 356.825,A -85,B 0,C 180,E1 -12444.382,E2 -12444.382} C_VEL
LIN {X 0,Y 374.493,Z 356.425,A -85,B 0,C 180,E1 -12445.736,E2 -12445.736} C_VEL
LIN {X 0,Y 374.522,Z 355.7,A -85,B 0,C 180,E1 -12446.767,E2 -12446.767} C_VEL
LIN {X 0,Y 374.616,Z 354.112,A -85,B 0,C 180,E1 -12448.146,E2 -12448.146} C_VEL
LIN {X 0,Y 374.857,Z 351.283,A -85,B 0,C 180,E1 -12449.79,E2 -12449.79} C_VEL
LIN {X 0,Y 375.107,Z 346.8,A -85,B 0,C 180,E1 -12451.641,E2 -12451.641} C_VEL
LIN {X 0,Y 375.576,Z 340.717,A -85,B 0,C 180,E1 -12453.505,E2 -12453.505} C_VEL
LIN {X 0,Y 375.993,Z 334.621,A -85,B 0,C 180,E1 -12454.978,E2 -12454.978} C_VEL
LIN {X 0,Y 376.703,Z 325.975,A -85,B 0,C 180,E1 -12456.656,E2 -12456.656} C_VEL
LIN {X 0,Y 377.264,Z 317.903,A -85,B 0,C 180,E1 -12457.933,E2 -12457.933} C_VEL
LIN {X 0,Y 378.021,Z 308.128,A -85,B 0,C 180,E1 -12459.206,E2 -12459.206} C_VEL
LIN {X 0,Y 378.775,Z 296.75,A -85,B 0,C 180,E1 -12460.391,E2 -12460.391} C_VEL
LIN {X 0,Y 379.478,Z 284.888,A -85,B 0,C 180,E1 -12461.371,E2 -12461.371} C_VEL
LIN {X 0,Y 380.11,Z 272.371,A -85,B 0,C 180,E1 -12462.153,E2 -12462.153} C_VEL
LIN {X 0,Y 380.488,Z 259.846,A -85,B 0,C 180,E1 -12462.724,E2 -12462.724} C_VEL
LIN {X 0,Y 380.878,Z 245.973,A -85,B 0,C 180,E1 -12463.124,E2 -12463.124} C_VEL
LIN {X 0,Y 382.444,Z 166.863,A -85,B 0,C 180,E1 -12464.847,E2 -12464.847} C_VEL
LIN {X 0,Y 379.872,Z 155.335,A -85,B 0,C 180,E1 -12465.226,E2 -12465.226} C_VEL
LIN {X 0,Y 376.709,Z 145.361,A -85,B 0,C 180,E1 -12465.604,E2 -12465.604} C_VEL
LIN {X 0,Y 376.026,Z 141.647,A -85,B 0,C 180,E1 -12466.569,E2 -12466.569} C_VEL
LIN {X 0,Y 375.96,Z 141.65,A -85,B 0,C 180,E1 -12470.537,E2 -12470.537} C_VEL
LIN {X 0,Y 375.963,Z 141.655,A -85,B 0,C 180,E1 -12473.495,E2 -12473.495} C_VEL
LIN {X 0,Y 375.959,Z 141.653,A -85,B 0,C 180,E1 -12475.888,E2 -12475.888} C_VEL
LIN {X 0,Y 375.964,Z 141.654,A -85,B 0,C 180,E1 -12479.687,E2 -12479.687} C_VEL
LIN {X 0,Y 375.995,Z 141.646,A -85,B 0,C 180,E1 -12482.141,E2 -12482.141} C_VEL
LIN {X 0,Y 376.006,Z 141.645,A -85,B 0,C 180,E1 -12484.539,E2 -12484.539} C_VEL
LIN {X 0,Y 375.962,Z 141.65,A -85,B 0,C 180,E1 -12488.045,E2 -12488.045} C_VEL
LIN {X 0,Y 376.001,Z 141.649,A -85,B 0,C 180,E1 -12491.472,E2 -12491.472} C_VEL
LIN {X 0,Y 376.057,Z 141.641,A -85,B 0,C 180,E1 -12494.832,E2 -12494.832} C_VEL
LIN {X 0,Y 376.049,Z 141.639,A -85,B 0,C 180,E1 -12498.136,E2 -12498.136} C_VEL
LIN {X 0,Y 376.217,Z 141.618,A -85,B 0,C 180,E1 -12501.919,E2 -12501.919} C_VEL
LIN {X 0,Y 376.168,Z 141.628,A -85,B 0,C 180,E1 -12504.639,E2 -12504.639} C_VEL
LIN {X 0,Y 376.333,Z 141.603,A -85,B 0,C 180,E1 -12508.028,E2 -12508.028} C_VEL
LIN {X 0,Y 376.488,Z 141.585,A -85,B 0,C 180,E1 -12510,E2 -12510} C_VEL
LIN {X 0,Y 376.25,Z 141.613,A -85,B 0,C 180,E1 -12512.694,E2 -12512.694} C_VEL
LIN {X 0,Y 375.496,Z 141.709,A -85,B 0,C 180,E1 -12513.587,E2 -12513.587} C_VEL
LIN {X 0,Y 372.619,Z 142.069,A -85,B 0,C 180,E1 -12515.039,E2 -12515.039} C_VEL
LIN {X 0,Y 370.242,Z 142.364,A -85,B 0,C 180,E1 -12516.213,E2 -12516.213} C_VEL
LIN {X 0,Y 369.235,Z 142.49,A -85,B 0,C 180,E1 -12517.121,E2 -12517.121} C_VEL
LIN {X 0,Y 369.156,Z 142.497,A -85,B 0,C 180,E1 -12517.428,E2 -12517.428} C_VEL
LIN {X 0,Y 369.02,Z 142.517,A -85,B 0,C 180,E1 -12520.979,E2 -12520.979} C_VEL
LIN {X 0,Y 369.013,Z 142.52,A -85,B 0,C 180,E1 -12524.335,E2 -12524.335} C_VEL
LIN {X 0,Y 368.998,Z 142.518,A -85,B 0,C 180,E1 -12527.768,E2 -12527.768} C_VEL
LIN {X 0,Y 368.907,Z 142.529,A -85,B 0,C 180,E1 -12531.221,E2 -12531.221} C_VEL
LIN {X 0,Y 368.952,Z 142.525,A -85,B 0,C 180,E1 -12534.775,E2 -12534.775} C_VEL
LIN {X 0,Y 368.968,Z 142.521,A -85,B 0,C 180,E1 -12537.203,E2 -12537.203} C_VEL
LIN {X 0,Y 368.921,Z 142.529,A -85,B 0,C 180,E1 -12539.689,E2 -12539.689} C_VEL
LIN {X 0,Y 368.898,Z 142.531,A -85,B 0,C 180,E1 -12543.537,E2 -12543.537} C_VEL
LIN {X 0,Y 368.899,Z 142.53,A -85,B 0,C 180,E1 -12546.856,E2 -12546.856} C_VEL
LIN {X 0,Y 368.949,Z 142.526,A -85,B 0,C 180,E1 -12550.364,E2 -12550.364} C_VEL
LIN {X 0,Y 368.955,Z 142.527,A -85,B 0,C 180,E1 -12553.628,E2 -12553.628} C_VEL
LIN {X 0,Y 368.903,Z 142.529,A -85,B 0,C 180,E1 -12556.699,E2 -12556.699} C_VEL
LIN {X 0,Y 368.949,Z 142.529,A -85,B 0,C 180,E1 -12559.635,E2 -12559.635} C_VEL
LIN {X 0,Y 368.899,Z 142.531,A -85,B 0,C 180,E1 -12563.144,E2 -12563.144} C_VEL
LIN {X 0,Y 368.894,Z 142.53,A -85,B 0,C 180,E1 -12566.462,E2 -12566.462} C_VEL
LIN {X 0,Y 368.925,Z 142.528,A -85,B 0,C 180,E1 -12569.047,E2 -12569.047} C_VEL
LIN {X 0,Y 368.976,Z 142.526,A -85,B 0,C 180,E1 -12571.564,E2 -12571.564} C_VEL
LIN {X 0,Y 368.997,Z 142.519,A -85,B 0,C 180,E1 -12574.02,E2 -12574.02} C_VEL
LIN {X 0,Y 368.929,Z 142.53,A -85,B 0,C 180,E1 -12577.605,E2 -12577.605} C_VEL
LIN {X 0,Y 368.98,Z 142.524,A -85,B 0,C 180,E1 -12581.107,E2 -12581.107} C_VEL
LIN {X 0,Y 368.995,Z 142.519,A -85,B 0,C 180,E1 -12584.535,E2 -12584.535} C_VEL
LIN {X 0,Y 369.002,Z 142.517,A -85,B 0,C 180,E1 -12587.907,E2 -12587.907} C_VEL
LIN {X 0,Y 369.185,Z 142.494,A -85,B 0,C 180,E1 -12591.846,E2 -12591.846} C_VEL
LIN {X 0,Y 369.14,Z 142.502,A -85,B 0,C 180,E1 -12594.538,E2 -12594.538} C_VEL
LIN {X 0,Y 369.317,Z 142.478,A -85,B 0,C 180,E1 -12597.819,E2 -12597.819} C_VEL
LIN {X 0,Y 369.456,Z 142.46,A -85,B 0,C 180,E1 -12600,E2 -12600} C_VEL
LIN {X 0,Y 369.317,Z 142.479,A -85,B 0,C 180,E1 -12602.182,E2 -12602.182} C_VEL
LIN {X 0,Y 369.207,Z 142.496,A -85,B 0,C 180,E1 -12606.559,E2 -12606.559} C_VEL
LIN {X 0,Y 369.136,Z 142.506,A -85,B 0,C 180,E1 -12608.761,E2 -12608.761} C_VEL
LIN {X 0,Y 369.004,Z 142.518,A -85,B 0,C 180,E1 -12612.094,E2 -12612.094} C_VEL
LIN {X 0,Y 368.997,Z 142.518,A -85,B 0,C 180,E1 -12615.465,E2 -12615.465} C_VEL
LIN {X 0,Y 368.982,Z 142.522,A -85,B 0,C 180,E1 -12618.893,E2 -12618.893} C_VEL
LIN {X 0,Y 368.922,Z 142.534,A -85,B 0,C 180,E1 -12622.396,E2 -12622.396} C_VEL
LIN {X 0,Y 368.998,Z 142.52,A -85,B 0,C 180,E1 -12625.981,E2 -12625.981} C_VEL
LIN {X 0,Y 368.96,Z 142.523,A -85,B 0,C 180,E1 -12628.812,E2 -12628.812} C_VEL
LIN {X 0,Y 368.898,Z 142.536,A -85,B 0,C 180,E1 -12632.238,E2 -12632.238} C_VEL
LIN {X 0,Y 368.929,Z 142.526,A -85,B 0,C 180,E1 -12635.002,E2 -12635.002} C_VEL
LIN {X 0,Y 368.912,Z 142.529,A -85,B 0,C 180,E1 -12638.642,E2 -12638.642} C_VEL
LIN {X 0,Y 368.91,Z 142.533,A -85,B 0,C 180,E1 -12641.819,E2 -12641.819} C_VEL
LIN {X 0,Y 368.88,Z 142.533,A -85,B 0,C 180,E1 -12645.177,E2 -12645.177} C_VEL
LIN {X 0,Y 368.883,Z 142.535,A -85,B 0,C 180,E1 -12648.178,E2 -12648.178} C_VEL
LIN {X 0,Y 368.908,Z 142.531,A -85,B 0,C 180,E1 -12651.36,E2 -12651.36} C_VEL
LIN {X 0,Y 368.937,Z 142.526,A -85,B 0,C 180,E1 -12655.147,E2 -12655.147} C_VEL
LIN {X 0,Y 368.93,Z 142.53,A -85,B 0,C 180,E1 -12659.047,E2 -12659.047} C_VEL
LIN {X 0,Y 368.95,Z 142.651,A -85,B 0,C 180,E1 -12659.881,E2 -12659.881} C_VEL
LIN {X 0,Y 371.836,Z 156.229,A -85,B 0,C 180,E1 -12663.024,E2 -12663.024} C_VEL
LIN {X 0,Y 372.587,Z 161.938,A -85,B 0,C 180,E1 -12664.289,E2 -12664.289} C_VEL
LIN {X 0,Y 371.048,Z 180.436,A -85,B 0,C 180,E1 -12668.142,E2 -12668.142} C_VEL
LIN {X 0,Y 370.768,Z 185.101,A -85,B 0,C 180,E1 -12669.112,E2 -12669.112} C_VEL
LIN {X 0,Y 375.043,Z 220.27,A -85,B 0,C 180,E1 -12670.131,E2 -12670.131} C_VEL
LIN {X 0,Y 373.571,Z 294.514,A -85,B 0,C 180,E1 -12671.81,E2 -12671.81} C_VEL
LIN {X 0,Y 372.908,Z 308.383,A -85,B 0,C 180,E1 -12672.344,E2 -12672.344} C_VEL
LIN {X 0,Y 372.117,Z 320.915,A -85,B 0,C 180,E1 -12673.049,E2 -12673.049} C_VEL
LIN {X 0,Y 371.241,Z 332.58,A -85,B 0,C 180,E1 -12673.927,E2 -12673.927} C_VEL
LIN {X 0,Y 370.451,Z 343.965,A -85,B 0,C 180,E1 -12675.021,E2 -12675.021} C_VEL
LIN {X 0,Y 369.636,Z 354.404,A -85,B 0,C 180,E1 -12676.276,E2 -12676.276} C_VEL
LIN {X 0,Y 368.99,Z 363.508,A -85,B 0,C 180,E1 -12677.628,E2 -12677.628} C_VEL
LIN {X 0,Y 368.248,Z 372.534,A -85,B 0,C 180,E1 -12679.276,E2 -12679.276} C_VEL
LIN {X 0,Y 367.855,Z 379.739,A -85,B 0,C 180,E1 -12680.932,E2 -12680.932} C_VEL
LIN {X 0,Y 367.675,Z 384.628,A -85,B 0,C 180,E1 -12682.311,E2 -12682.311} C_VEL
LIN {X 0,Y 367.537,Z 389.144,A -85,B 0,C 180,E1 -12683.904,E2 -12683.904} C_VEL
LIN {X 0,Y 367.55,Z 392.796,A -85,B 0,C 180,E1 -12685.614,E2 -12685.614} C_VEL
LIN {X 0,Y 367.504,Z 394.511,A -85,B 0,C 180,E1 -12686.712,E2 -12686.712} C_VEL
LIN {X 0,Y 367.629,Z 395.807,A -85,B 0,C 180,E1 -12687.809,E2 -12687.809} C_VEL
LIN {X 0,Y 367.603,Z 396.672,A -85,B 0,C 180,E1 -12688.905,E2 -12688.905} C_VEL
LIN {X 0,Y 367.594,Z 397.073,A -85,B 0,C 180,E1 -12690,E2 -12690} C_VEL
LIN {X 0,Y 367.583,Z 397.045,A -85,B 0,C 180,E1 -12691.096,E2 -12691.096} C_VEL
LIN {X 0,Y 367.528,Z 396.607,A -85,B 0,C 180,E1 -12692.192,E2 -12692.192} C_VEL
LIN {X 0,Y 367.452,Z 395.753,A -85,B 0,C 180,E1 -12693.29,E2 -12693.29} C_VEL
LIN {X 0,Y 367.478,Z 394.437,A -85,B 0,C 180,E1 -12694.388,E2 -12694.388} C_VEL
LIN {X 0,Y 367.415,Z 391.914,A -85,B 0,C 180,E1 -12695.916,E2 -12695.916} C_VEL
LIN {X 0,Y 367.663,Z 387.833,A -85,B 0,C 180,E1 -12697.69,E2 -12697.69} C_VEL
LIN {X 0,Y 367.965,Z 382.87,A -85,B 0,C 180,E1 -12699.344,E2 -12699.344} C_VEL
LIN {X 0,Y 368.639,Z 375.463,A -85,B 0,C 180,E1 -12701.269,E2 -12701.269} C_VEL
LIN {X 0,Y 369.537,Z 367.446,A -85,B 0,C 180,E1 -12702.913,E2 -12702.913} C_VEL
LIN {X 0,Y 370.51,Z 357.853,A -85,B 0,C 180,E1 -12704.496,E2 -12704.496} C_VEL
LIN {X 0,Y 371.588,Z 348.29,A -85,B 0,C 180,E1 -12705.777,E2 -12705.777} C_VEL
LIN {X 0,Y 372.86,Z 337.054,A -85,B 0,C 180,E1 -12706.988,E2 -12706.988} C_VEL
LIN {X 0,Y 374.251,Z 324.453,A -85,B 0,C 180,E1 -12708.051,E2 -12708.051} C_VEL
LIN {X 0,Y 375.257,Z 312.219,A -85,B 0,C 180,E1 -12708.849,E2 -12708.849} C_VEL
LIN {X 0,Y 376.398,Z 297.957,A -85,B 0,C 180,E1 -12709.497,E2 -12709.497} C_VEL
LIN {X 0,Y 376.957,Z 284.67,A -85,B 0,C 180,E1 -12709.893,E2 -12709.893} C_VEL
LIN {X 0,Y 378.724,Z 220.11,A -85,B 0,C 180,E1 -12711.413,E2 -12711.413} C_VEL
LIN {X 0,Y 376.798,Z 204.706,A -85,B 0,C 180,E1 -12711.969,E2 -12711.969} C_VEL
LIN {X 0,Y 373.421,Z 186.438,A -85,B 0,C 180,E1 -12712.748,E2 -12712.748} C_VEL
LIN {X 0,Y 372.327,Z 181.242,A -85,B 0,C 180,E1 -12712.998,E2 -12712.998} C_VEL
LIN {X 0,Y 373.919,Z 165.967,A -85,B 0,C 180,E1 -12716.212,E2 -12716.212} C_VEL
LIN {X 0,Y 373.821,Z 163.285,A -85,B 0,C 180,E1 -12716.822,E2 -12716.822} C_VEL
LIN {X 0,Y 371.754,Z 153.501,A -85,B 0,C 180,E1 -12719.245,E2 -12719.245} C_VEL
LIN {X 0,Y 368.926,Z 142.534,A -85,B 0,C 180,E1 -12722.236,E2 -12722.236} C_VEL
LIN {X 0,Y 368.933,Z 142.531,A -85,B 0,C 180,E1 -12725.001,E2 -12725.001} C_VEL
LIN {X 0,Y 368.913,Z 142.532,A -85,B 0,C 180,E1 -12728.64,E2 -12728.64} C_VEL
LIN {X 0,Y 368.885,Z 142.535,A -85,B 0,C 180,E1 -12732.009,E2 -12732.009} C_VEL
LIN {X 0,Y 368.883,Z 142.535,A -85,B 0,C 180,E1 -12735.176,E2 -12735.176} C_VEL
LIN {X 0,Y 368.886,Z 142.53,A -85,B 0,C 180,E1 -12738.178,E2 -12738.178} C_VEL
LIN {X 0,Y 368.91,Z 142.525,A -85,B 0,C 180,E1 -12741.36,E2 -12741.36} C_VEL
LIN {X 0,Y 368.94,Z 142.526,A -85,B 0,C 180,E1 -12745.146,E2 -12745.146} C_VEL
LIN {X 0,Y 368.933,Z 142.523,A -85,B 0,C 180,E1 -12749.046,E2 -12749.046} C_VEL
LIN {X 0,Y 368.966,Z 142.525,A -85,B 0,C 180,E1 -12752.796,E2 -12752.796} C_VEL
LIN {X 0,Y 368.949,Z 142.525,A -85,B 0,C 180,E1 -12756.113,E2 -12756.113} C_VEL
LIN {X 0,Y 368.939,Z 142.525,A -85,B 0,C 180,E1 -12759.947,E2 -12759.947} C_VEL
LIN {X 0,Y 368.972,Z 142.524,A -85,B 0,C 180,E1 -12763.398,E2 -12763.398} C_VEL
LIN {X 0,Y 369.061,Z 142.511,A -85,B 0,C 180,E1 -12766.79,E2 -12766.79} C_VEL
LIN {X 0,Y 369.066,Z 142.514,A -85,B 0,C 180,E1 -12770.131,E2 -12770.131} C_VEL
LIN {X 0,Y 369.176,Z 142.503,A -85,B 0,C 180,E1 -12773.441,E2 -12773.441} C_VEL
LIN {X 0,Y 369.317,Z 142.486,A -85,B 0,C 180,E1 -12777.818,E2 -12777.818} C_VEL
LIN {X 0,Y 369.44,Z 142.645,A -85,B 0,C 180,E1 -12780.068,E2 -12780.068} C_VEL
LIN {X 0,Y 370.937,Z 149.229,A -85,B 0,C 180,E1 -12781.951,E2 -12781.951} C_VEL
LIN {X 0,Y 379.413,Z 168.508,A -85,B 0,C 180,E1 -12783.229,E2 -12783.229} C_VEL
LIN {X 0,Y 379.998,Z 171.322,A -85,B 0,C 180,E1 -12783.354,E2 -12783.354} C_VEL
LIN {X 0,Y 377.344,Z 255.947,A -85,B 0,C 180,E1 -12785.376,E2 -12785.376} C_VEL
LIN {X 0,Y 376.782,Z 268.922,A -85,B 0,C 180,E1 -12785.888,E2 -12785.888} C_VEL
LIN {X 0,Y 375.98,Z 282.259,A -85,B 0,C 180,E1 -12786.649,E2 -12786.649} C_VEL
LIN {X 0,Y 375.015,Z 293.854,A -85,B 0,C 180,E1 -12787.538,E2 -12787.538} C_VEL
LIN {X 0,Y 373.952,Z 305.19,A -85,B 0,C 180,E1 -12788.647,E2 -12788.647} C_VEL
LIN {X 0,Y 372.955,Z 314.419,A -85,B 0,C 180,E1 -12789.764,E2 -12789.764} C_VEL
LIN {X 0,Y 371.872,Z 323.888,A -85,B 0,C 180,E1 -12791.169,E2 -12791.169} C_VEL
LIN {X 0,Y 370.721,Z 333.083,A -85,B 0,C 180,E1 -12792.87,E2 -12792.87} C_VEL
LIN {X 0,Y 369.91,Z 339.342,A -85,B 0,C 180,E1 -12794.312,E2 -12794.312} C_VEL
LIN {X 0,Y 369.167,Z 345.312,A -85,B 0,C 180,E1 -12796.024,E2 -12796.024} C_VEL
LIN {X 0,Y 368.58,Z 349.969,A -85,B 0,C 180,E1 -12797.763,E2 -12797.763} C_VEL
LIN {X 0,Y 368.247,Z 352.406,A -85,B 0,C 180,E1 -12798.932,E2 -12798.932} C_VEL
LIN {X 0,Y 367.863,Z 354.976,A -85,B 0,C 180,E1 -12800.586,E2 -12800.586} C_VEL
LIN {X 0,Y 367.588,Z 356.724,A -85,B 0,C 180,E1 -12802.481,E2 -12802.481} C_VEL
LIN {X 0,Y 367.478,Z 357.18,A -85,B 0,C 180,E1 -12803.679,E2 -12803.679} C_VEL
LIN {X 0,Y 367.42,Z 357.126,A -85,B 0,C 180,E1 -12804.886,E2 -12804.886} C_VEL
LIN {X 0,Y 367.423,Z 356.597,A -85,B 0,C 180,E1 -12806.1,E2 -12806.1} C_VEL
LIN {X 0,Y 367.451,Z 355.497,A -85,B 0,C 180,E1 -12807.324,E2 -12807.324} C_VEL
LIN {X 0,Y 367.669,Z 352.858,A -85,B 0,C 180,E1 -12809.172,E2 -12809.172} C_VEL
LIN {X 0,Y 367.975,Z 348.889,A -85,B 0,C 180,E1 -12811.042,E2 -12811.042} C_VEL
LIN {X 0,Y 368.307,Z 343.47,A -85,B 0,C 180,E1 -12812.901,E2 -12812.901} C_VEL
LIN {X 0,Y 368.796,Z 337.338,A -85,B 0,C 180,E1 -12814.536,E2 -12814.536} C_VEL
LIN {X 0,Y 369.366,Z 329.836,A -85,B 0,C 180,E1 -12816.145,E2 -12816.145} C_VEL
LIN {X 0,Y 369.997,Z 321.483,A -85,B 0,C 180,E1 -12817.604,E2 -12817.604} C_VEL
LIN {X 0,Y 370.778,Z 311.586,A -85,B 0,C 180,E1 -12819,E2 -12819} C_VEL
LIN {X 0,Y 371.515,Z 301.159,A -85,B 0,C 180,E1 -12820.193,E2 -12820.193} C_VEL
LIN {X 0,Y 372.265,Z 290.044,A -85,B 0,C 180,E1 -12821.216,E2 -12821.216} C_VEL
LIN {X 0,Y 372.916,Z 277.903,A -85,B 0,C 180,E1 -12822.083,E2 -12822.083} C_VEL
LIN {X 0,Y 373.472,Z 264.064,A -85,B 0,C 180,E1 -12822.812,E2 -12822.812} C_VEL
LIN {X 0,Y 373.883,Z 251.142,A -85,B 0,C 180,E1 -12823.257,E2 -12823.257} C_VEL
LIN {X 0,Y 375.594,Z 167.647,A -85,B 0,C 180,E1 -12825.126,E2 -12825.126} C_VEL
LIN {X 0,Y 373.125,Z 156.969,A -85,B 0,C 180,E1 -12825.489,E2 -12825.489} C_VEL
LIN {X 0,Y 369.572,Z 145.653,A -85,B 0,C 180,E1 -12825.943,E2 -12825.943} C_VEL
LIN {X 0,Y 368.958,Z 142.527,A -85,B 0,C 180,E1 -12826.793,E2 -12826.793} C_VEL
LIN {X 0,Y 368.911,Z 142.534,A -85,B 0,C 180,E1 -12829.642,E2 -12829.642} C_VEL
LIN {X 0,Y 368.9,Z 142.532,A -85,B 0,C 180,E1 -12833.144,E2 -12833.144} C_VEL
LIN {X 0,Y 368.895,Z 142.53,A -85,B 0,C 180,E1 -12836.461,E2 -12836.461} C_VEL
LIN {X 0,Y 368.928,Z 142.528,A -85,B 0,C 180,E1 -12839.046,E2 -12839.046} C_VEL
LIN {X 0,Y 368.979,Z 142.525,A -85,B 0,C 180,E1 -12841.563,E2 -12841.563} C_VEL
LIN {X 0,Y 368.999,Z 142.518,A -85,B 0,C 180,E1 -12844.019,E2 -12844.019} C_VEL
LIN {X 0,Y 368.932,Z 142.529,A -85,B 0,C 180,E1 -12847.604,E2 -12847.604} C_VEL
LIN {X 0,Y 368.953,Z 142.528,A -85,B 0,C 180,E1 -12851.105,E2 -12851.105} C_VEL
LIN {X 0,Y 368.996,Z 142.519,A -85,B 0,C 180,E1 -12854.535,E2 -12854.535} C_VEL
LIN {X 0,Y 369.004,Z 142.517,A -85,B 0,C 180,E1 -12857.906,E2 -12857.906} C_VEL
LIN {X 0,Y 369.186,Z 142.494,A -85,B 0,C 180,E1 -12861.846,E2 -12861.846} C_VEL
LIN {X 0,Y 369.14,Z 142.502,A -85,B 0,C 180,E1 -12864.537,E2 -12864.537} C_VEL
LIN {X 0,Y 369.318,Z 142.478,A -85,B 0,C 180,E1 -12867.818,E2 -12867.818} C_VEL
LIN {X 0,Y 369.457,Z 142.46,A -85,B 0,C 180,E1 -12870,E2 -12870} C_VEL
